(* CODESYS project CtaAppFU_1.0.0.2.library
   Description: FU Library der CTA
   Version: 1.0.0.2
   Title: CtaAppFU
   Author: SIS
   DocFormat: reStructuredText
   LanguageModelAttribute: qualified-access-only
   Placeholder: CtaAppFU
   DefaultNamespace: CtaAppFU
   CompiledLibraryCompatibilityVersion: CODESYS V3.5 SP16 Patch 3
   Company: CTA

Project tree, tasks and I/O mapping:
  libraries: Standard, 3.5.18.0 (System); CtaAppBasic, 1.0.0.0 (CTA); CtaAppBmk, 1.0.0.0 (CTA); CtaAppReport, 1.0.0.2 (CTA); CtaSysConfig, 1.0.0.2 (CTA); VisuDialogs, 3.5.16.20 (System); VisuSymbols, 4.5.0.0 (System); CtaSysFU, 1.0.0.0 (CTA); CtaAppTime, 1.0.0.1 (CTA); CtaVisSymbols, 1.0.0.0 (CTA); CtaAppInfluxLog, 1.0.0.0 (CTA); CtaSysBase, 1.0.0.0 (CTA); CtaAppWagoModbus, 1.0.0.0 (CTA); CtaAppModbus, 1.0.0.0 (CTA)
  40 Visualizations/
    ABB/
      580/
        visualisation DIA_ABB580
        TABLE/
          visualisation VIS_FU_ABB_TABLE
        VISU/
          visualisation VIS_ABB580
          visualisation VIS_ABB580_QUERY
      880/
        TABLE/
          visualisation VIS_FU_ABB_TABLE_880
        VISU/
          visualisation VIS_ABB880
          visualisation VIS_ABB880_QUERY
        visualisation DIA_ABB880
    BITZER/
      CSV/
        TABLE/
          visualisation VIS_FU_BITZER_TABLE
        VISU/
          visualisation VIS_BITZER_CSV
          visualisation VIS_BITZER_CSV_QUERY
        visualisation DIA_BITZER_CSV
  00000000-0000-0000-0000-000000000000|D:\CoDeSys\LibrariesV3\trunk\Intern\CAA\CAA Template\3.4.0.0 draft\Placeholder.xml
  00000000-0000-0000-0000-000000000000|D:\CoDeSys\LibrariesV3\trunk\Intern\CAA\CAA Template\3.2.0.3 draft\Prefix.pdf
  00000000-0000-0000-0000-000000000000|D:\CoDeSys\LibrariesV3\trunk\Intern\CAA\CAA Template\3.5.2.0 draft\Placeholder.xml
  20 Structs/
    Modbus/
      data type scParameter
      data type scModBus
    ABB/
      580/
        data type scFuAbb580Table
      880/
        data type scFuAbb880Table
    BITZER/
      CSV/
        data type enEnvelopeZone
        data type enEnvelopeState
        data type scFuBitzerCSVTable
        data type enFuState
  50 Images/
  10 Documenation/
    global variables VersionHistory
    global variables readMe
  21 Interface/
    ABB/
      880/
        interface ITF_FU_ABB_880: proayscTable
      580/
        interface ITF_FU_ABB_580: proayscTable
    BITZER/
      CSV/
        interface ITF_FU_BITZER_CSV: proayscTable
  11 Library Parameter/
    global variables Parameter
  12 Konstanten/
    global variables GlobalKonstant
  60 Textlisten/
    ABB 580/
      text list Error_ABB580_880
      text list Info_ABB580_880
      text list Warnung_ABB580_880
      text list FU_ABB_580_880_PARA
    BITZER/
      text list Error_BITZER_CSV
      text list Info_BITZER_CSV
      text list Warnung_BITZER_CSV
      text list FU_BITZER_CSV_PARA
  13 Globale Variablen/
    global variables GVL_FU
  text list GlobalTextList
  5ce3da45-db07-42e7-a21c-a00fff4ed8f6|C:\Users\sis\Downloads\dip-switch.svg
  5ce3da45-db07-42e7-a21c-a00fff4ed8f6|C:\Users\sis\Downloads\lightning-bolt-circle.svg
  30 Program Organization Units/
    ABB/
      580/
        function block FB_FU_ABB580 [ST]: proFU_TYPE, FB_INIT, COM_DATA, actCwSw, metParIdToMbAdr, metHzScaleFromFU, metHzScaleToFU, actCheckFirmWare, actCheckLastComCall, actTrendLog, actReport, actConfig, actTable, proayscTable
      880/
        function block FB_FU_ABB880 [ST]: FB_INIT, proFU_TYPE, COM_DATA, actCwSw, metParIdToMbAdr, metHzScaleFromFU, metHzScaleToFU, actCheckFirmWare, actCheckLastComCall, actTrendLog, actReport, actConfig, actTable, proayscTable
    Bitzer/
      CSV/
        function block FB_FU_BITZER_CSV [ST]: FB_INIT, COM_DATA, actCwSw, actCheckFirmWare, actCheckLastComCall, actTrendLog, actReport, actConfig, actTable, proayscTable, proFU_TYPE
  5ce3da45-db07-42e7-a21c-a00fff4ed8f6|C:\Users\sis\Downloads\sine-wave.svg
  5ce3da45-db07-42e7-a21c-a00fff4ed8f6|C:\Users\sis\Downloads\eye.svg
  5ce3da45-db07-42e7-a21c-a00fff4ed8f6|C:\Users\sis\Downloads\lan.svg
*)

// 20 Structs/Modbus/scParameter
TYPE scParameter :
	STRUCT
		scModBus	:	scModBus;
	END_STRUCT
END_TYPE

// 20 Structs/Modbus/scModBus
TYPE scModBus :
	STRUCT
		fbxMbErrorAsWarning	:	CtaSysConfig.fbBOOL;
	END_STRUCT
END_TYPE

// 20 Structs/ABB/580/scFuAbb580Table
TYPE scFuAbb580Table :
	STRUCT
		stParaNr		:	STRING(5);
		stValue			:	STRING(20);
	END_STRUCT
END_TYPE

// 20 Structs/ABB/880/scFuAbb880Table
TYPE scFuAbb880Table :
	STRUCT
		stParaNr		:	STRING(5);
		stValue			:	STRING(20);
	END_STRUCT
END_TYPE

// 20 Structs/BITZER/CSV/enEnvelopeZone
{attribute 'to_string'}
TYPE enEnvelopeZone :
	(
		inside 				:= 	0,
		SST_Low_SDT_Low		:=	1,
		SST_Low				:=	2,
		SST_Low_SDT_High	:=	3,
		SDT_High			:=	4,
		SST_High_SDT_High	:=	5,
		SST_High			:=	6,
		SST_High_SDT_Low	:=	7,
		SDT_Low				:= 	8	
	);
END_TYPE

// 20 Structs/BITZER/CSV/enEnvelopeState
{attribute 'to_string'}
TYPE enEnvelopeState :
	(
		stopped 	:= 0,
		starting 	:= 1,
		running		:= 2,
		stopping	:= 3,
		warning		:= 4,
		critical	:= 5,
		fault		:= 6,
		defrosting	:= 7
	);
END_TYPE

// 20 Structs/BITZER/CSV/scFuBitzerCSVTable
TYPE scFuBitzerCSVTable :
	STRUCT
		stParaNr		:	STRING(5);
		stValue			:	STRING(20);
	END_STRUCT
END_TYPE

// 20 Structs/BITZER/CSV/enFuState
{attribute 'to_string'}
TYPE enFuState :
	(
		not_ready		:=	0,
		power_not_ready :=	1,
		stopped			:=	2,
		short_Cycling	:=	3,
		start_Delay		:=	4,
		freeze			:=	5,
		running			:=	6,
		DC_Inj			:=	7,
		stopping		:=	8,
		locked			:=	9,
		fault			:= 10,
		service			:= 11
	);
END_TYPE

// 10 Documenation/VersionHistory
(* 

.. image:: ../../Images/CTA_Logo.jpg
   :align: right
   :width: 15% 

**Vorlage**   


============ =========== =========== ============================================
**Date**     **Version** **Author**  **Change**
------------ ----------- ----------- --------------------------------------------
04.03.2021   0.0.0.0     SIS         Vorlage erstellt

============ =========== =========== ============================================


*)
VAR_GLOBAL
    stInfo : STRING:= '0.0.0.0, Vorlage, CTA';
END_VAR

// 10 Documenation/readMe
(*

**ReadMe**
 
|	**Empfehlung**
|
|	Bibliothek CtaAppFU zur dämpfung und rampung von Signalen
|	Instanzieren Sie den CtaAppFU.fbFU in ihrem Funktionsbaustein oder POU beispielsweise als fbFUx ( x = Nr. des FU's 
|	Deklarieren Sie die Struktur Variable welche als Parameter und zur ansteuerung dienen wie im Code beispiel.
|  
| *Beispiel* 

+-----------------------+---------------------------------------------------------------------------------------------------------------------------------------------------------------------------------------------------------------------------------------------------------------------------------------------------------------------------------------------------------------------------------------------------------------------------------------+
| Beschreibung          |  Code                                                                                                                                                                                                                                                                                                                                                                                                                                 |
+=======================+=======================================================================================================================================================================================================================================================================================================================================================================================================================================+
| POU oder SmFb         | .. code-block:: codesys                                                                                                                                                                                                                                                                                                                                                                                                               |
|                       |                                                                                                                                                                                                                                                                                                                                                                                                                                       |
|                       |	// Deklaration als VAR im POU oder dem selbsterstellten Funktionsbaustein                                                                                                                                                                                                                                                                                                                                                        	|
|                       |   VAR   																																																				 																																																				|
|						|	    (*Frequenzumformer 1*)																																																		 																																																	|
|						|		fbFU1			: CtaAppFU.fbFU;																																																																																																|
|			 			|	END_VAR                                                                                                                                                                                                                                                                                                                                                                                                                          	|
+-----------------------+---------------------------------------------------------------------------------------------------------------------------------------------------------------------------------------------------------------------------------------------------------------------------------------------------------------------------------------------------------------------------------------------------------------------------------------+
| Code für Init         | .. code-block:: codesys                                                                                                                                                                                                                                                                                                                                                                                                               |
|                       |   																																																					 																																																				|
|			 			|	// Kopieren des nachfolgenden Codes in eine Action zur Initialisierung der Parameter. Zum Beispiel actConfig.																																																				 																										|
|                       |	{region "Parameter Temperaturfühler 1"}                                                                                                                                                                                                                                                                                                                                                                                             |
|			 			|		(*Basis*)                                                                                                                                                                                                                                                                                                                                                                                                                       |
|						|		fbFU1.scParameter.scModBus.fbxMbErrorAsWarning					(_WertInit := FALSE																	 	 		);     //P1 Parameter zur behandlung eines ModBus Fehlers als Warnung.																																															|
|						|	{endregion}                                                                                                                                                      																																																																    | 
|						|																																																																																																										|
+-----------------------+---------------------------------------------------------------------------------------------------------------------------------------------------------------------------------------------------------------------------------------------------------------------------------------------------------------------------------------------------------------------------------------------------------------------------------------+
*)                                                                                                                                                                                                                                                                                                                                                                                                                                                               
VAR_GLOBAL
	xReadMeDone              :   BOOL; 
END_VAR

// 13 Globale Variablen/GVL_FU
{attribute 'qualified_only'}
VAR_GLOBAL

END_VAR

// 11 Library Parameter/Parameter
{attribute 'qualified_only'}
VAR_GLOBAL CONSTANT
 	stABB580_FirmWare	:	STRING(20) := '2.20.0.12';
	stABB880_FirmWare	:	STRING(20) := '3.46.0.03';
	stBITZER_FirmWare	:	STRING(20) := '2.15.0.10';
END_VAR

// 12 Konstanten/GlobalKonstant
{attribute 'qualified_only'}
VAR_GLOBAL CONSTANT 	
	stReportTextListErrorAbb580_880   	: CtaAppReport.stReportTextList := 'CtaAppFU.Error_ABB580_880';
	stReportTextListWarningAbb580_880 	: CtaAppReport.stReportTextList := 'CtaAppFU.Warnung_ABB580_880';
	stReportTextListInfoAbb580_880  	: CtaAppReport.stReportTextList := 'CtaAppFU.Info_ABB580_880';
	stReportTextListErrorBitzerCsv   	: CtaAppReport.stReportTextList := 'CtaAppFU.Error_BITZER_CSV';
	stReportTextListWarningBitzerCsv 	: CtaAppReport.stReportTextList := 'CtaAppFU.Warnung_BITZER_CSV';
	stReportTextListInfoBitzerCsv    	: CtaAppReport.stReportTextList := 'CtaAppFU.Info_BITZER_CSV';		
END_VAR

// 30 Program Organization Units/ABB/580/FB_FU_ABB580
FUNCTION_BLOCK FB_FU_ABB580 EXTENDS CtaSysFU.FB_FU_BASE IMPLEMENTS ITF_FU_ABB_580
VAR_INPUT
END_VAR
VAR_OUTPUT
END_VAR
VAR
	(* Case *)
	iCaseCw					: 	INT;
	(* BUS Controll *)
	xResetAfterInit 		:   BOOL	:= TRUE;
	{attribute 'displaymode':='hex'}
	wControllWord   		:   WORD;
    wSollwert       		:   WORD;
	{attribute 'displaymode':='hex'}
    wStateWord      		:   WORD;
    wIstwert        		:   WORD;	
	xLocRemError			:	BOOL;
	(* HZ Scale Faktor *)
	rScaleFaktorHzMax   	:   REAL;    
    rScaleFaktorHzMin   	:   REAL;
	(* Energy Zähler *)
	uiGWhCount  			:   UINT;
    uiMWhCount  			:   UINT;
    uiKWhCount  			:   UINT;      
	(* Code from FU *)
	{attribute 'displaymode':='hex'}
	wErrorAkt       		:   WORD;
	{attribute 'displaymode':='hex'}
	wErrorOld1      		:   WORD;     
	{attribute 'displaymode':='hex'}   
	wErrorOld2      		:   WORD;    
	rHzOnError				:	REAL; 
	rTempOnError			:	REAL;
	(* Report*)     	
	iError					: 	INT;    
    difor					:	DINT;                                                                    
    ayErrorReporter			:	ARRAY[20..25] OF CtaAppReport.fbReporter;
	ayWarningReporter		:	ARRAY[20..25] OF CtaAppReport.fbReporter;	
	(* Trend Log *)
	fbTrendrAmpere			:	CtaAppInfluxLog.FB_LOG_NODE_REAL;
	fbTrendrVolt			:	CtaAppInfluxLog.FB_LOG_NODE_REAL;
	fbTrendrHz				:	CtaAppInfluxLog.FB_LOG_NODE_REAL;
	fbTrendrkW				:	CtaAppInfluxLog.FB_LOG_NODE_REAL;
	fbTrendrTemperatur		:	CtaAppInfluxLog.FB_LOG_NODE_REAL;
	fbTrendxError			:	CtaAppInfluxLog.FB_LOG_NODE_BOOL;
	fbTrendrGwh				:	CtaAppInfluxLog.FB_LOG_NODE_REAL;
	fbTrendrMwh				:	CtaAppInfluxLog.FB_LOG_NODE_REAL;
	fbTrendrkwh				:	CtaAppInfluxLog.FB_LOG_NODE_REAL;
	(* Modbus *)
	stVendorName			:	STRING(20);
	stMajorMinorRevision	:	STRING(20);
	xFirmWareOK				:	BOOL;
	fbLastComDataCall		:	CtaAppTime.fbTimeMeasurement;
	ltLastComCall			:	LTIME;
	xAccesOk				:	BOOL;
	xModbusOk				:	BOOL;
	aywTempRead				:	ARRAY[0..16] OF WORD;
	(* Tabelle *)
	ayscTable				:	ARRAY[0..16] OF scFuAbb580Table;
	(* Config *)
	fbConfigFile			:	CtaSysConfig.fbConfigFile;	
	scParameter				:	scParameter;
END_VAR

(* Config *)
actConfig();
(* Check Firmware *)
actCheckFirmWare();
(* Check Last Acces *)
actCheckLastComCall();
(* Controll & State Word *)
actCwSw();
(* Trend Log *)
actTrendLog();
(* Table *)
actTable();
(* Report *)
actReport();

PROPERTY proFU_TYPE : STRING(20)
GET
proFU_TYPE := 'ABB 580';
END_GET
END_PROPERTY

//FB_Init ist immer implizit verfügbar und wird primär für die Initialisierung verwendet.
//Der Rückgabewert wird nicht ausgewertet. Für gezielte Einflussnahme können Sie
//die Methoden explizit deklarieren und darin mit dem Standard-Initialisierungscode 
//zusätzlichen Code bereitstellen. Sie können den Rückgabewert auswerten.
METHOD FB_Init: BOOL
VAR_INPUT    
bInitRetains: BOOL; // TRUE: Die Retain-Variablen werden initialisiert (Reset warm / Reset kalt)    
bInCopyCode: BOOL;  // TRUE: Die Instanz wird danach in den Kopiercode kopiert (Online-Change)
END_VAR
SUPER^.stVisuDiaName := 'CtaAppFU.DIA_ABB580';
END_METHOD

METHOD COM_DATA
VAR_INPUT
	ITF_MB_CLIENT		:	CtaSysBase.ITF_BASE;
END_VAR
VAR
	ITF_MB_CLIENT_WAGO	: 	CtaAppWagoModbus.ITF_MbClient;
	ITF_MB_CLIENT_CS	:	CtaAppModbus.ITF_CLIENT;
END_VAR
IF __QUERYINTERFACE(ITF_MB_CLIENT,ITF_MB_CLIENT_WAGO) THEN
	(* COM DATA Call *)
	fbLastComDataCall.Start();
	(* Client Info *)
	ITF_MB_CLIENT_WAGO.metITF_BMK(THIS^);
	stVendorName 				:= ITF_MB_CLIENT_WAGO.sVendorName;
	stMajorMinorRevision 		:= ITF_MB_CLIENT_WAGO.sMajorMinorRevision;
	xModbusOk 					:= ITF_MB_CLIENT_WAGO.proModBusOK;
	(*-Modbus Fc----------------------------------------------------------------------------------------Umrechnung------------------------------------------------------------------------------------------Kommentar-------*)
	(* Fc3 *)	
	ITF_MB_CLIENT_WAGO.metFc3ReadHoldingRegister		(metParIdToMbAdr(00,04),ADR(aywTempRead[ 0])	,1,0);	wStateWord					:= aywTempRead[ 0];														// Parameter 00.04 Adr.    3	Status Word
	ITF_MB_CLIENT_WAGO.metFc3ReadHoldingRegister		(metParIdToMbAdr(00,05),ADR(aywTempRead[ 1])	,1,0);	wIstwert					:= aywTempRead[ 1];														// Parameter 00.05 Adr.    4	Status Wert
	ITF_MB_CLIENT_WAGO.metFc3ReadHoldingRegister		(metParIdToMbAdr(01,06),ADR(aywTempRead[ 2])	,1,0);	rAcknowledge_Hz				:= metHzScaleFromFU(aywTempRead[ 2],rScaleFaktorHzMax);					// Parameter 01.06 Adr.  105	Aktuelle Hz							
	ITF_MB_CLIENT_WAGO.metFc3ReadHoldingRegister		(metParIdToMbAdr(01,07),ADR(aywTempRead[ 3])	,1,0);  rAmpere						:= TO_REAL(aywTempRead[ 3])	/ 10;										// Parameter 01.07 Adr.  106	Aktuelle Ampere                                                               									
	ITF_MB_CLIENT_WAGO.metFc3ReadHoldingRegister		(metParIdToMbAdr(01,13),ADR(aywTempRead[ 4])	,1,0);	rVolt						:= aywTempRead[ 4];														// Parameter 01.13 Adr.  112	Aktuelle Spannung                                                                                               									
	ITF_MB_CLIENT_WAGO.metFc3ReadHoldingRegister		(metParIdToMbAdr(01,14),ADR(aywTempRead[ 5])	,1,0);	rkWatt						:= TO_REAL(aywTempRead[ 5])	/ 10;										// Parameter 01.14 Adr.  113	Aktuelle Leistung kW
	ITF_MB_CLIENT_WAGO.metFc3ReadHoldingRegister		(metParIdToMbAdr(01,18),ADR(aywTempRead[ 6])	,1,0);	uiGWhCount					:= aywTempRead[ 6];														// Parameter 01.18 Adr.  117	Leistung GWh
	ITF_MB_CLIENT_WAGO.metFc3ReadHoldingRegister		(metParIdToMbAdr(01,19),ADR(aywTempRead[ 7])	,1,0);	uiMWhCount					:= aywTempRead[ 7];														// Parameter 01.19 Adr.  118	Leistung MWh	
	ITF_MB_CLIENT_WAGO.metFc3ReadHoldingRegister		(metParIdToMbAdr(01,20),ADR(aywTempRead[ 8])	,1,0);	uiKWhCount					:= TO_UINT(aywTempRead[ 8])  / 10;										// Parameter 01.20 Adr.  119	Leistung KWh	
	ITF_MB_CLIENT_WAGO.metFc3ReadHoldingRegister		(metParIdToMbAdr(04,01),ADR(aywTempRead[ 9])	,1,0);	wErrorAkt					:= aywTempRead[ 9];														// Parameter 04.01 Adr.  400	Aktueller Fehler
	ITF_MB_CLIENT_WAGO.metFc3ReadHoldingRegister		(metParIdToMbAdr(04,02),ADR(aywTempRead[10])	,1,0);	wErrorOld1					:= aywTempRead[10];														// Parameter 04.02 Adr.  401	Letzter Fehler
	ITF_MB_CLIENT_WAGO.metFc3ReadHoldingRegister		(metParIdToMbAdr(04,03),ADR(aywTempRead[11])	,1,0);	wErrorOld2					:= aywTempRead[11];														// Parameter 04.03 Adr.  402	Vorletzter Fehler
	ITF_MB_CLIENT_WAGO.metFc3ReadHoldingRegister		(metParIdToMbAdr(05,10),ADR(aywTempRead[12])	,1,0);	rTemperatur					:= aywTempRead[12];														// Parameter 05.10 Adr.  509	Temperatur
(* Modbusprobleme Parameter Existieren nicht mehr 14.10.2024 SIS *)
//	ITF_MB_CLIENT_WAGO.metFc3ReadHoldingRegister		(metParIdToMbAdr(05,81),ADR(aywTempRead[13])	,1,0);	rHzOnError					:= metHzScaleFromFU(aywTempRead[13],rScaleFaktorHzMax);					// Parameter 05.81 Adr.  580	Frequenz bei Fehler
//	ITF_MB_CLIENT_WAGO.metFc3ReadHoldingRegister		(metParIdToMbAdr(05,87),ADR(aywTempRead[14])	,1,0);	rTempOnError				:= aywTempRead[14];														// Parameter 05.87 Adr.  586	Temperatur bei Fehler
	
	ITF_MB_CLIENT_WAGO.metFc3ReadHoldingRegister		(metParIdToMbAdr(30,13),ADR(aywTempRead[15])	,1,0);	rScaleFaktorHzMin			:= metHzScaleFromFU(aywTempRead[15],rScaleFaktorHzMax);					// Parameter 30.13 Adr. 3012	Min Hz Skalierfaktor
	ITF_MB_CLIENT_WAGO.metFc3ReadHoldingRegister		(metParIdToMbAdr(46,02),ADR(aywTempRead[16])	,1,0);	rScaleFaktorHzMax			:= TO_REAL(aywTempRead[16])  / 10;										// Parameter 46.02 Adr. 4600	Max Hz Skalierfaktor
	                                                                                                                        		                                                    					
	(*  Fc16 *)                                                                                             	        														        					
	ITF_MB_CLIENT_WAGO.metFc16WriteHoldingRegisters	(metParIdToMbAdr(00,01),ADR(wControllWord)		,1,0);  																									// Parameter 00.01 Adr.   0	Controll Word
	ITF_MB_CLIENT_WAGO.metFc16WriteHoldingRegisters	(metParIdToMbAdr(00,02),ADR(wSollwert)			,1,0);  																									// Parameter 00.02 Adr.   1	Soll Wert
ELSIF __QUERYINTERFACE(ITF_MB_CLIENT,ITF_MB_CLIENT_CS) THEN
	(* COM DATA Call *)
	fbLastComDataCall.Start();
	ITF_MB_CLIENT_CS.CREATE_JOB	( 3, metParIdToMbAdr(00,04),ADR(aywTempRead[ 0])	,1);	wStateWord					:= aywTempRead[ 0];														// Parameter 00.04 Adr.    3	Status Word
	ITF_MB_CLIENT_CS.CREATE_JOB ( 3, metParIdToMbAdr(00,05),ADR(aywTempRead[ 1])	,1);	wIstwert					:= aywTempRead[ 1];														// Parameter 00.05 Adr.    4	Status Wert
	ITF_MB_CLIENT_CS.CREATE_JOB ( 3, metParIdToMbAdr(01,06),ADR(aywTempRead[ 2])	,1);	rAcknowledge_Hz				:= metHzScaleFromFU(aywTempRead[ 2],rScaleFaktorHzMax);					// Parameter 01.06 Adr.  105	Aktuelle Hz							
	ITF_MB_CLIENT_CS.CREATE_JOB ( 3, metParIdToMbAdr(01,07),ADR(aywTempRead[ 3])	,1);  	rAmpere						:= TO_REAL(aywTempRead[ 3])	/ 10;										// Parameter 01.07 Adr.  106	Aktuelle Ampere                                  
	ITF_MB_CLIENT_CS.CREATE_JOB ( 3, metParIdToMbAdr(01,13),ADR(aywTempRead[ 4])	,1);	rVolt						:= aywTempRead[ 4];														// Parameter 01.13 Adr.  112	Aktuelle Spannung                                
	ITF_MB_CLIENT_CS.CREATE_JOB ( 3, metParIdToMbAdr(01,14),ADR(aywTempRead[ 5])	,1);	rkWatt						:= TO_REAL(aywTempRead[ 5])	/ 10;										// Parameter 01.14 Adr.  113	Aktuelle Leistung kW
	ITF_MB_CLIENT_CS.CREATE_JOB	( 3, metParIdToMbAdr(01,18),ADR(aywTempRead[ 6])	,1);	uiGWhCount					:= aywTempRead[ 6];														// Parameter 01.18 Adr.  117	Leistung GWh
	ITF_MB_CLIENT_CS.CREATE_JOB	( 3, metParIdToMbAdr(01,19),ADR(aywTempRead[ 7])	,1);	uiMWhCount					:= aywTempRead[ 7];														// Parameter 01.19 Adr.  118	Leistung MWh	
	ITF_MB_CLIENT_CS.CREATE_JOB	( 3, metParIdToMbAdr(01,20),ADR(aywTempRead[ 8])	,1);	uiKWhCount					:= TO_UINT(aywTempRead[ 8])  / 10;										// Parameter 01.20 Adr.  119	Leistung KWh	
	ITF_MB_CLIENT_CS.CREATE_JOB	( 3, metParIdToMbAdr(04,01),ADR(aywTempRead[ 9])	,1);	wErrorAkt					:= aywTempRead[ 9];														// Parameter 04.01 Adr.  400	Aktueller Fehler
	ITF_MB_CLIENT_CS.CREATE_JOB	( 3, metParIdToMbAdr(04,02),ADR(aywTempRead[10])	,1);	wErrorOld1					:= aywTempRead[10];														// Parameter 04.02 Adr.  401	Letzter Fehler
	ITF_MB_CLIENT_CS.CREATE_JOB	( 3, metParIdToMbAdr(04,03),ADR(aywTempRead[11])	,1);	wErrorOld2					:= aywTempRead[11];														// Parameter 04.03 Adr.  402	Vorletzter Fehler
	ITF_MB_CLIENT_CS.CREATE_JOB	( 3, metParIdToMbAdr(05,10),ADR(aywTempRead[12])	,1);	rTemperatur					:= aywTempRead[12];														// Parameter 05.10 Adr.  509	Temperatur
(* Modbusprobleme Parameter Existieren nicht mehr 14.10.2024 SIS *)
//	ITF_MB_CLIENT_CS.CREATE_JOB	( 3, metParIdToMbAdr(05,81),ADR(aywTempRead[13])	,1);	rHzOnError					:= metHzScaleFromFU(aywTempRead[13],rScaleFaktorHzMax);					// Parameter 05.81 Adr.  580	Frequenz bei Fehler
//	ITF_MB_CLIENT_CS.CREATE_JOB	( 3, metParIdToMbAdr(05,87),ADR(aywTempRead[14])	,1);	rTempOnError				:= aywTempRead[14];														// Parameter 05.87 Adr.  586	Temperatur bei Fehler
	
	ITF_MB_CLIENT_CS.CREATE_JOB	( 3, metParIdToMbAdr(30,13),ADR(aywTempRead[15])	,1);	rScaleFaktorHzMin			:= metHzScaleFromFU(aywTempRead[15],rScaleFaktorHzMax);					// Parameter 30.13 Adr. 3012	Min Hz Skalierfaktor
	ITF_MB_CLIENT_CS.CREATE_JOB	( 3, metParIdToMbAdr(46,02),ADR(aywTempRead[16])	,1);	rScaleFaktorHzMax			:= TO_REAL(aywTempRead[16])  / 10;										// Parameter 46.02 Adr. 4600	Max Hz Skalierfaktor

	(*  Fc16 *)                                                                                             	        														        					
	ITF_MB_CLIENT_CS.CREATE_JOB	(16, metParIdToMbAdr(00,01),ADR(wControllWord)		,1);  																									// Parameter 00.01 Adr.   0	Controll Word
	ITF_MB_CLIENT_CS.CREATE_JOB	(16, metParIdToMbAdr(00,02),ADR(wSollwert)			,1);  				
	xModbusOk := NOT ITF_MB_CLIENT_CS.ERROR;
	stVendorName := 'ABB';
	stMajorMinorRevision := Parameter.stABB580_FirmWare;
ELSE
	xModbusOk := FALSE;	
END_IF
xBusOK := xModbusOk;
END_METHOD

ACTION actCwSw:
(*--Controll Word-------------------------------------------State Word-----------------*)(*          
    wControllWord.0  = Aus1                                 wStateWord.0      = RDY_ON       
    wControllWord.1  = Aus2                                 wStateWord.1      = RDY_RUN      
    wControllWord.2  = Aus3                                 wStateWord.2      = RDY_REF      
    wControllWord.3  = Inhibit_Operation                    wStateWord.3      = TRIPPED      
    wControllWord.4  = Rampenausgang_Null                   wStateWord.4      = OFF_2_STATUS 
    wControllWord.5  = Rampenausgang_Halten                 wStateWord.5      = OFF_3_STATUS 
    wControllWord.6  = Rampeneingang_Null                   wStateWord.6      = SWC_ON_INHIB 
    wControllWord.7  = Quittierung                          wStateWord.7      = ALARM        
    wControllWord.8  = Jogging_1                            wStateWord.8      = AUF_SOLLWERT 
    wControllWord.9  = Jogginng_2                           wStateWord.9      = REMOTE       
    wControllWord.10 = Fernsteuerung                        wStateWord.10     = ÜBER_LIMIT   
    wControllWord.11 = EXT_CTRL_LOC                         wStateWord.11     = USER_0       
    wControllWord.12 = USER_0                               wStateWord.12     = USER_1       
    wControllWord.13 = USER_1                               wStateWord.13     = USER_2       
    wControllWord.14 = USER_2                               wStateWord.14     = USER_3       
    wControllWord.15 = USER_3                             	wStateWord.15     = RESERVE *)   
    
	   (* Quittieren *)
		wControllWord.7 := wStateWord.9 AND (xResetAfterInit 	 OR (ayErrorReporter[20].metGetQuitt() 
																 OR  ayErrorReporter[21].metGetQuitt() 
																 OR  ayErrorReporter[22].metGetQuitt() 
																 OR  ayErrorReporter[23].metGetQuitt()
																 OR  ayErrorReporter[24].metGetQuitt()
																 OR  ayErrorReporter[25].metGetQuitt()) 
																 OR xQuitt); 
		(* Status Werte *)
		xReady          := wStateWord.1 AND wStateWord.9;
		IF NOT xResetAfterInit THEN
			xLocRemError    := NOT wStateWord.9;
			xHandLockal		:= xLocRemError;
			xAcknowledge    := wStateWord.8; // OR wStateWord0616.14
			xError      	:= wStateWord.3;   
		END_IF;
		(* Bei Störmeldung oder Initialisierung in Case 0 Springen *)   
		IF xError THEN
			iCaseCw         := 0;   
		END_IF;   
		IF xReady THEN
			xResetAfterInit := FALSE;
		END_IF;
		(* Sollwert *)
		wSollwert := INT_TO_WORD(LIMIT(WORD_TO_INT(metHzScaleToFU(rScaleFaktorHzMin,rScaleFaktorHzMax)),WORD_TO_INT(metHzScaleToFU(rRelease_Hz,rScaleFaktorHzMax)),WORD_TO_INT(metHzScaleToFU(rScaleFaktorHzMax,rScaleFaktorHzMax)))); 
		(* FU Steuerung *)
		CASE iCaseCw OF
			0: // Nicht Einschaltbereit
				// Start Value 
				wControllWord.1  := TRUE;       // Nicht Aus 2 
				wControllWord.2  := TRUE;       // Nicht Aus 3 
				wControllWord.3  := FALSE;
				wControllWord.10 := TRUE;       // Steuerung Bus
				// Statusabfrage Nicht Einschaltbereit 
				wControllWord.0 := FALSE; 
				iCaseCw := iCaseCw + 1;   
			1: // Einschaltbereit           
				IF NOT wStateWord.1 AND NOT wStateWord.0 THEN      
					wControllWord.0 := FALSE;   
				ELSIF wStateWord.0 THEN 
					wControllWord.0 := TRUE; 
				END_IF;
				IF wStateWord.1 AND wStateWord.0 THEN                      
					iCaseCw := iCaseCw + 1;        
				END_IF;          
			2: // Betriebsbereit
				IF NOT xRelease AND NOT wStateWord.1 THEN
					iCaseCw := 0;
				END_IF;
				// Freigabe
				wControllWord.3 := xRelease;        
				// Wenn Betrieb Freigegeben weiter
				IF wStateWord.2 THEN
					IF wControllWord.3 THEN
						wControllWord.4 := TRUE;
						wControllWord.5 := TRUE;
						wControllWord.6 := TRUE;
						iCaseCw := iCaseCw + 1; 
					ELSE
						iCaseCw := 1;
					END_IF;
				END_IF;
			3: // Betrieb Freigegeben
				// Freigabe
				wControllWord.3 := xRelease AND iError = 0; 
				wControllWord.0 := xRelease AND iError = 0; 
				IF wControllWord.3 THEN
					wControllWord.4 := TRUE;
					wControllWord.5 := TRUE;
					wControllWord.6 := TRUE;
				ELSE
					iCaseCw := 0;
				END_IF;  
		ELSE
			iCaseCw := 0;           
		END_CASE;
END_ACTION

METHOD PRIVATE metParIdToMbAdr : WORD
VAR_INPUT
    usiMainParaId   :   USINT;
    usiSubParaId    :   USINT;
END_VAR
metParIdToMbAdr := (usiMainParaId * 100) + usiSubParaId - 1;
END_METHOD

METHOD PRIVATE metHzScaleFromFU : REAL
VAR_INPUT
    wModBusValue   :    WORD;
    rScaleFaktor   :    REAL;
END_VAR
VAR
	iModBusValue	:	INT;
END_VAR
iModBusValue := TO_INT(wModBusValue);
metHzScaleFromFU := rScaleFaktor / 20000 * TO_REAL(iModBusValue);
END_METHOD

METHOD PRIVATE metHzScaleToFU : WORD
VAR_INPUT
    rValue         :    REAL;
    rScaleFaktor   :    REAL;
END_VAR
rScaleFaktor := LIMIT(0,rScaleFaktor,65535);
IF rScaleFaktor <> 0 THEN
    metHzScaleToFU := TO_WORD(TO_INT(20000 / rScaleFaktor * rValue));
ELSE
    metHzScaleToFU := 0;
END_IF;
END_METHOD

ACTION actCheckFirmWare:
(* Check Firmware *)
IF FIND(stVendorName,'ABB') <> 0 THEN
	IF FIND(stMajorMinorRevision,Parameter.stABB580_FirmWare) <> 0 THEN
		xFirmWareOK := TRUE;	
	ELSE
		xFirmWareOK := FALSE;
	END_IF
ELSE
	xFirmWareOK := FALSE;
END_IF
END_ACTION

ACTION actCheckLastComCall:
(* Last Acces *)
ltLastComCall := fbLastComDataCall.Stop();
IF ltLastComCall <= LTIME#2S AND ltLastComCall >LTIME#0NS THEN
	xAccesOk := TRUE;
ELSE
	xAccesOk := FALSE;	
END_IF;
END_ACTION

ACTION actTrendLog:
(* Ampere *)
fbTrendrAmpere.ENABLE			:= TRUE;
fbTrendrAmpere.KEY				:= CONCAT(stObjID,'_rAmpere');
fbTrendrAmpere.SET_VALUE		:= rAmpere;

(* Volt *)
fbTrendrVolt.ENABLE				:= TRUE;
fbTrendrVolt.KEY				:= CONCAT(stObjID,'_rVolt');
fbTrendrVolt.SET_VALUE			:= rVolt;

(* HZ *)
fbTrendrHz.ENABLE				:= TRUE;
fbTrendrHz.KEY					:= CONCAT(stObjID,'_rHZ');
fbTrendrHz.SET_VALUE			:= rAcknowledge_Hz;

(* kW *)
fbTrendrkW.ENABLE				:= TRUE;
fbTrendrkW.KEY					:= CONCAT(stObjID,'_rkW');
fbTrendrkW.SET_VALUE			:= rkWatt;

(* Temperatur *)
fbTrendrTemperatur.ENABLE		:= TRUE;
fbTrendrTemperatur.KEY			:= CONCAT(stObjID,'_rTemperatur');
fbTrendrTemperatur.SET_VALUE	:= rTemperatur;

(* Error *)
fbTrendxError.ENABLE			:= TRUE;
fbTrendxError.KEY				:= CONCAT(stObjID,'_xError');
fbTrendxError.SET_VALUE			:= xError;

(* Gwh *)
fbTrendrGwh.ENABLE				:= TRUE;
fbTrendrGwh.KEY					:= CONCAT(stObjID,'_rGwh');
fbTrendrGwh.SET_VALUE			:= uiGWhCount;

(* Mwh *)
fbTrendrMwh.ENABLE				:= TRUE;
fbTrendrMwh.KEY					:= CONCAT(stObjID,'_rMwh');
fbTrendrMwh.SET_VALUE			:= uiMWhCount;

(* kwh *)
fbTrendrkwh.ENABLE				:= TRUE;
fbTrendrkwh.KEY					:= CONCAT(stObjID,'_rkwh');
fbTrendrkwh.SET_VALUE			:= uiKWhCount;
END_ACTION

ACTION actReport:
IF __QUERYINTERFACE(ITF_REPORTMANAGER,ITF_REPORTMANAGER) THEN

(* Errors *)                        
	(* Meldung Modbus Error *)
	ayErrorReporter[20].proPrio  := 1;
	ayErrorReporter[20].metReport(     		xSetReportIn					:= NOT xModbusOk AND xEnable,
											iReportID						:= 20,
											enReportTypeIn					:= SEL(scParameter.scModBus.fbxMbErrorAsWarning.xValue,CtaAppReport.enReportType.Error,CtaAppReport.enReportType.Warning),  
											enReportAcknowledgeTypeIn   	:= CtaAppReport.enReportacknowledgeType.Auto,
											tDelay							:= T#4S, 
											ITF_BMK_IN						:= THIS^,			              
											pstReportTextListIn				:= ADR(GlobalKonstant.stReportTextListErrorAbb580_880),
											stOptionalReportText		    := '',   
											iRetryTilReportLock 		    := 0, 
											xResetCount         		    := FALSE,  
											tReset						    := T#24H); 		

	(* Meldung Modbus Software Zugriff Fehler *)
	ayErrorReporter[21].proPrio  := 1;
	ayErrorReporter[21].metReport(     		xSetReportIn					:= NOT xAccesOk AND xEnable,
											iReportID						:= 21,
											enReportTypeIn					:= SEL(scParameter.scModBus.fbxMbErrorAsWarning.xValue,CtaAppReport.enReportType.Error,CtaAppReport.enReportType.Warning),  
											enReportAcknowledgeTypeIn   	:= CtaAppReport.enReportacknowledgeType.Auto,
											tDelay							:= T#4S, 
											ITF_BMK_IN						:= THIS^,			              
											pstReportTextListIn				:= ADR(GlobalKonstant.stReportTextListErrorAbb580_880),
											stOptionalReportText		    := '',   
											iRetryTilReportLock 		    := 0, 
											xResetCount         		    := FALSE,  
											tReset						    := T#24H); 		

	(* Meldung FU Error *)
	ayErrorReporter[22].proPrio  := 1;
	ayErrorReporter[22].metReport(     		xSetReportIn					:= xError AND xEnable,
											iReportID						:= 22,
											enReportTypeIn					:= CtaAppReport.enReportType.Error,  
											enReportAcknowledgeTypeIn   	:= CtaAppReport.enReportacknowledgeType.QUIT,
											tDelay							:= T#4S, 
											ITF_BMK_IN						:= THIS^,			              
											pstReportTextListIn				:= ADR(GlobalKonstant.stReportTextListErrorAbb580_880),
											stOptionalReportText		    := CtaAppReport.fcWordToHexString(wErrorAkt),   
											iRetryTilReportLock 		    := 0, 
											xResetCount         		    := FALSE,  
											tReset						    := T#24H); 	
											
	(* Meldung Firmware Missmatch *)
	ayWarningReporter[20].proPrio  := 1;
	ayWarningReporter[20].metReport(     	xSetReportIn					:= NOT xFirmWareOK AND xEnable,
											iReportID						:= 20,
											enReportTypeIn					:= CtaAppReport.enReportType.Warning,  
											enReportAcknowledgeTypeIn   	:= CtaAppReport.enReportacknowledgeType.Auto,
											tDelay							:= T#4S, 
											ITF_BMK_IN						:= THIS^,			              
											pstReportTextListIn				:= ADR(GlobalKonstant.stReportTextListWarningAbb580_880),
											stOptionalReportText		    := Parameter.stABB580_FirmWare,   
											iRetryTilReportLock 		    := 0, 
											xResetCount         		    := FALSE,  
											tReset						    := T#24H); 	
											
	(* Sync Reports *)                                         
	FOR difor := LOWER_BOUND(ayErrorReporter,1) TO UPPER_BOUND(ayErrorReporter,1) DO
		ITF_REPORTMANAGER.metSyncReporter(ayErrorReporter[difor]);	
	END_FOR;
	FOR difor := LOWER_BOUND(ayWarningReporter,1) TO UPPER_BOUND(ayWarningReporter,1) DO
		ITF_REPORTMANAGER.metSyncReporter(ayWarningReporter[difor]);	
	END_FOR;


END_IF;
END_ACTION

ACTION actConfig:
fbConfigFile();

scParameter.scModBus.fbxMbErrorAsWarning(_usiParaNr	:= 1, itfConfigFb := fbConfigFile);
END_ACTION

ACTION actTable:
ayscTable[00].stParaNr	:= 	'00.04';
ayscTable[00].stValue	:=	TO_STRING(CtaAppReport.fcWordToHexString(wStateWord));

ayscTable[01].stParaNr	:= 	'00.05';
ayscTable[01].stValue	:=	TO_STRING(wIstwert);

ayscTable[02].stParaNr	:= 	'01.06';
ayscTable[02].stValue	:=	CONCAT(TO_STRING(rAcknowledge_Hz),' Hz');

ayscTable[03].stParaNr	:= 	'01.07';
ayscTable[03].stValue	:=	CONCAT(TO_STRING(rAmpere),' A');

ayscTable[04].stParaNr	:= 	'01.13';
ayscTable[04].stValue	:=	CONCAT(TO_STRING(rVolt),' V');

ayscTable[05].stParaNr	:= 	'01.14';
ayscTable[05].stValue	:=	CONCAT(TO_STRING(rkWatt),' kW');

ayscTable[06].stParaNr	:= 	'01.18';
ayscTable[06].stValue	:=	CONCAT(TO_STRING(uiGWhCount),' GWh');

ayscTable[07].stParaNr	:= 	'01.19';
ayscTable[07].stValue	:=	CONCAT(TO_STRING(uiMWhCount),' MWh');

ayscTable[08].stParaNr	:= 	'01.20';
ayscTable[08].stValue	:=	CONCAT(TO_STRING(uiKWhCount),' KWh');

ayscTable[09].stParaNr	:= 	'04.01';
ayscTable[09].stValue	:=	TO_STRING(CtaAppReport.fcWordToHexString(wErrorAkt));

ayscTable[10].stParaNr	:= 	'04.02';
ayscTable[10].stValue	:=	TO_STRING(CtaAppReport.fcWordToHexString(wErrorOld1));

ayscTable[11].stParaNr	:= 	'04.03';
ayscTable[11].stValue	:=	TO_STRING(CtaAppReport.fcWordToHexString(wErrorOld2));

ayscTable[12].stParaNr	:= 	'05.10';
ayscTable[12].stValue	:=	CONCAT(TO_STRING(rTemperatur),' °C');

ayscTable[13].stParaNr	:= 	'05.81';
ayscTable[13].stValue	:=	CONCAT(TO_STRING(rHzOnError),' Hz');

ayscTable[14].stParaNr	:= 	'05.87';
ayscTable[14].stValue	:=	CONCAT(TO_STRING(rTempOnError),' °C');

ayscTable[15].stParaNr	:= 	'30.13';
ayscTable[15].stValue	:=	CONCAT(TO_STRING(rScaleFaktorHzMin),' Hz');

ayscTable[16].stParaNr	:= 	'46.02';
ayscTable[16].stValue	:=	CONCAT(TO_STRING(rScaleFaktorHzMax),' Hz');
END_ACTION

PROPERTY proayscTable : ARRAY[0..16] OF scFuAbb580Table;
GET
proayscTable := ayscTable;
END_GET
END_PROPERTY

END_FUNCTION_BLOCK

// 21 Interface/ABB/580/ITF_FU_ABB_580
INTERFACE ITF_FU_ABB_580 EXTENDS CtaSysFU.ITF_FU_BASE

PROPERTY proayscTable : ARRAY[0..16] OF scFuAbb580Table;
GET
END_GET
END_PROPERTY

END_INTERFACE

// 30 Program Organization Units/ABB/880/FB_FU_ABB880
FUNCTION_BLOCK FB_FU_ABB880 EXTENDS CtaSysFU.FB_FU_BASE IMPLEMENTS ITF_FU_ABB_880
VAR_INPUT
END_VAR
VAR_OUTPUT
END_VAR
VAR
	(* Case *)
	iCaseCw					: 	INT;
	(* BUS Controll *)
	xResetAfterInit 		:   BOOL	:= TRUE;
	{attribute 'displaymode':='hex'}
	wControllWord   		:   WORD;
    wSollwert       		:   WORD;
	{attribute 'displaymode':='hex'}
    wStateWord      		:   WORD;
    wIstwert        		:   WORD;	
	xLocRemError			:	BOOL;
	(* HZ Scale Faktor *)
	rScaleFaktorHzMax   	:   REAL;    
    rScaleFaktorHzMin   	:   REAL;
	(* Energy Zähler *)
	uiGWhCount  			:   UINT;
    uiMWhCount  			:   UINT;
    uiKWhCount  			:   UINT;      
	(* Code from FU *)
	{attribute 'displaymode':='hex'}
	wErrorAkt       		:   WORD;
	{attribute 'displaymode':='hex'}
	wErrorOld1      		:   WORD;     
	{attribute 'displaymode':='hex'}   
	wErrorOld2      		:   WORD;    
	rHzOnError				:	REAL; 
	rTempOnError			:	REAL;
	(* Report*)     	
	iError					: 	INT;    
    difor					:	DINT;                                                                    
    ayErrorReporter			:	ARRAY[20..25] OF CtaAppReport.fbReporter;
	ayWarningReporter		:	ARRAY[20..25] OF CtaAppReport.fbReporter;	
	(* Trend Log *)
    fbTrendrAmpere			:	CtaAppInfluxLog.FB_LOG_NODE_REAL;
	fbTrendrVolt			:	CtaAppInfluxLog.FB_LOG_NODE_REAL;
	fbTrendrHz				:	CtaAppInfluxLog.FB_LOG_NODE_REAL;
	fbTrendrkW				:	CtaAppInfluxLog.FB_LOG_NODE_REAL;
	fbTrendrTemperatur		:	CtaAppInfluxLog.FB_LOG_NODE_REAL;
	fbTrendxError			:	CtaAppInfluxLog.FB_LOG_NODE_BOOL;
	fbTrendrGwh				:	CtaAppInfluxLog.FB_LOG_NODE_REAL;
	fbTrendrMwh				:	CtaAppInfluxLog.FB_LOG_NODE_REAL;
	fbTrendrkwh				:	CtaAppInfluxLog.FB_LOG_NODE_REAL;
	(* Modbus *)
	stVendorName			:	STRING(20);
	stMajorMinorRevision	:	STRING(20);
	xFirmWareOK				:	BOOL;
	fbLastComDataCall		:	CtaAppTime.fbTimeMeasurement;
	ltLastComCall			:	LTIME;
	xAccesOk				:	BOOL;
	xModbusOk				:	BOOL;
	aywTempRead				:	ARRAY[0..16] OF WORD;
	(* Tabelle *)
	ayscTable				:	ARRAY[0..16] OF scFuAbb880Table;
	(* Config *)
	fbConfigFile			:	CtaSysConfig.fbConfigFile;	
	scParameter				:	scParameter;
END_VAR

(* Config *)
actConfig();
(* Check Firmware *)
actCheckFirmWare();
(* Check Last Acces *)
actCheckLastComCall();
(* Controll & State Word *)
actCwSw();
(* Trend Log *)
actTrendLog();
(* Table *)
actTable();
(* Report *)
actReport();

//FB_Init ist immer implizit verfügbar und wird primär für die Initialisierung verwendet.
//Der Rückgabewert wird nicht ausgewertet. Für gezielte Einflussnahme können Sie
//die Methoden explizit deklarieren und darin mit dem Standard-Initialisierungscode 
//zusätzlichen Code bereitstellen. Sie können den Rückgabewert auswerten.
METHOD FB_Init: BOOL
VAR_INPUT    
bInitRetains: BOOL; // TRUE: Die Retain-Variablen werden initialisiert (Reset warm / Reset kalt)    
bInCopyCode: BOOL;  // TRUE: Die Instanz wird danach in den Kopiercode kopiert (Online-Change)
END_VAR
SUPER^.stVisuDiaName := 'CtaAppFU.DIA_ABB880';
END_METHOD

PROPERTY proFU_TYPE : STRING(20)
GET
proFU_TYPE := 'ABB 880';
END_GET
END_PROPERTY

METHOD COM_DATA
VAR_INPUT
	ITF_MB_CLIENT		:	CtaSysBase.ITF_BASE;
END_VAR
VAR
	ITF_MB_CLIENT_WAGO	: 	CtaAppWagoModbus.ITF_MbClient;
	ITF_MB_CLIENT_CS	:	CtaAppModbus.ITF_CLIENT;
END_VAR
IF __QUERYINTERFACE(ITF_MB_CLIENT,ITF_MB_CLIENT_WAGO) THEN
	(* COM DATA Call *)
	fbLastComDataCall.Start();
	(* Client Info *)
	ITF_MB_CLIENT_WAGO.metITF_BMK(THIS^);
	stVendorName 				:= ITF_MB_CLIENT_WAGO.sVendorName;
	stMajorMinorRevision 		:= ITF_MB_CLIENT_WAGO.sMajorMinorRevision;
	xModbusOk 					:= ITF_MB_CLIENT_WAGO.proModBusOK;
	(*-Modbus Fc----------------------------------------------------------------------------------------Umrechnung------------------------------------------------------------------------------------------Kommentar-------*)
	(* Fc3 *)	
	ITF_MB_CLIENT_WAGO.metFc3ReadHoldingRegister		(metParIdToMbAdr(00,04),ADR(aywTempRead[ 0])	,1,0);	wStateWord					:= aywTempRead[ 0];														// Parameter 00.04 Adr.    3	Status Word
	ITF_MB_CLIENT_WAGO.metFc3ReadHoldingRegister		(metParIdToMbAdr(00,05),ADR(aywTempRead[ 1])	,1,0);	wIstwert					:= aywTempRead[ 1];														// Parameter 00.05 Adr.    4	Status Wert
	ITF_MB_CLIENT_WAGO.metFc3ReadHoldingRegister		(metParIdToMbAdr(01,06),ADR(aywTempRead[ 2])	,1,0);	rAcknowledge_Hz				:= metHzScaleFromFU(aywTempRead[ 2],rScaleFaktorHzMax);					// Parameter 01.06 Adr.  105	Aktuelle Hz							
	ITF_MB_CLIENT_WAGO.metFc3ReadHoldingRegister		(metParIdToMbAdr(01,07),ADR(aywTempRead[ 3])	,1,0);  rAmpere						:= TO_REAL(aywTempRead[ 3])	/ 10;										// Parameter 01.07 Adr.  106	Aktuelle Ampere                                                               									
	ITF_MB_CLIENT_WAGO.metFc3ReadHoldingRegister		(metParIdToMbAdr(01,13),ADR(aywTempRead[ 4])	,1,0);	rVolt						:= aywTempRead[ 4];														// Parameter 01.13 Adr.  112	Aktuelle Spannung                                                                                               									
	ITF_MB_CLIENT_WAGO.metFc3ReadHoldingRegister		(metParIdToMbAdr(01,14),ADR(aywTempRead[ 5])	,1,0);	rkWatt						:= TO_REAL(aywTempRead[ 5])	/ 10;										// Parameter 01.14 Adr.  113	Aktuelle Leistung kW
	ITF_MB_CLIENT_WAGO.metFc3ReadHoldingRegister		(metParIdToMbAdr(01,18),ADR(aywTempRead[ 6])	,1,0);	uiGWhCount					:= aywTempRead[ 6];														// Parameter 01.18 Adr.  117	Leistung GWh
	ITF_MB_CLIENT_WAGO.metFc3ReadHoldingRegister		(metParIdToMbAdr(01,19),ADR(aywTempRead[ 7])	,1,0);	uiMWhCount					:= aywTempRead[ 7];														// Parameter 01.19 Adr.  118	Leistung MWh	
	ITF_MB_CLIENT_WAGO.metFc3ReadHoldingRegister		(metParIdToMbAdr(01,20),ADR(aywTempRead[ 8])	,1,0);	uiKWhCount					:= TO_UINT(aywTempRead[ 8])  / 10;										// Parameter 01.20 Adr.  119	Leistung KWh	
	ITF_MB_CLIENT_WAGO.metFc3ReadHoldingRegister		(metParIdToMbAdr(04,01),ADR(aywTempRead[ 9])	,1,0);	wErrorAkt					:= aywTempRead[ 9];														// Parameter 04.01 Adr.  400	Aktueller Fehler
	ITF_MB_CLIENT_WAGO.metFc3ReadHoldingRegister		(metParIdToMbAdr(04,02),ADR(aywTempRead[10])	,1,0);	wErrorOld1					:= aywTempRead[10];														// Parameter 04.02 Adr.  401	Letzter Fehler
	ITF_MB_CLIENT_WAGO.metFc3ReadHoldingRegister		(metParIdToMbAdr(04,03),ADR(aywTempRead[11])	,1,0);	wErrorOld2					:= aywTempRead[11];														// Parameter 04.03 Adr.  402	Vorletzter Fehler
	ITF_MB_CLIENT_WAGO.metFc3ReadHoldingRegister		(metParIdToMbAdr(05,10),ADR(aywTempRead[12])	,1,0);	rTemperatur					:= aywTempRead[12];														// Parameter 05.10 Adr.  509	Temperatur
(* Modbusprobleme Parameter Existieren nicht mehr 14.10.2024 SIS *)
//	ITF_MB_CLIENT_WAGO.metFc3ReadHoldingRegister		(metParIdToMbAdr(05,81),ADR(aywTempRead[13])	,1,0);	rHzOnError					:= metHzScaleFromFU(aywTempRead[13],rScaleFaktorHzMax);					// Parameter 05.81 Adr.  580	Frequenz bei Fehler
//	ITF_MB_CLIENT_WAGO.metFc3ReadHoldingRegister		(metParIdToMbAdr(05,87),ADR(aywTempRead[14])	,1,0);	rTempOnError				:= aywTempRead[14];														// Parameter 05.87 Adr.  586	Temperatur bei Fehler
	
	ITF_MB_CLIENT_WAGO.metFc3ReadHoldingRegister		(metParIdToMbAdr(30,13),ADR(aywTempRead[15])	,1,0);	rScaleFaktorHzMin			:= metHzScaleFromFU(aywTempRead[15],rScaleFaktorHzMax);					// Parameter 30.13 Adr. 3012	Min Hz Skalierfaktor
	ITF_MB_CLIENT_WAGO.metFc3ReadHoldingRegister		(metParIdToMbAdr(46,02),ADR(aywTempRead[16])	,1,0);	rScaleFaktorHzMax			:= TO_REAL(aywTempRead[16])  / 10;										// Parameter 46.02 Adr. 4600	Max Hz Skalierfaktor
	                                                                                                                        		                                                    					
	(*  Fc16 *)                                                                                             	        														        					
	ITF_MB_CLIENT_WAGO.metFc16WriteHoldingRegisters	(metParIdToMbAdr(00,01),ADR(wControllWord)		,1,0);  																									// Parameter 00.01 Adr.   0	Controll Word
	ITF_MB_CLIENT_WAGO.metFc16WriteHoldingRegisters	(metParIdToMbAdr(00,02),ADR(wSollwert)			,1,0);  																									// Parameter 00.02 Adr.   1	Soll Wert
ELSIF __QUERYINTERFACE(ITF_MB_CLIENT,ITF_MB_CLIENT_CS) THEN
	(* COM DATA Call *)
	fbLastComDataCall.Start();
	ITF_MB_CLIENT_CS.CREATE_JOB	( 3, metParIdToMbAdr(00,04),ADR(aywTempRead[ 0])	,1);	wStateWord					:= aywTempRead[ 0];														// Parameter 00.04 Adr.    3	Status Word
	ITF_MB_CLIENT_CS.CREATE_JOB ( 3, metParIdToMbAdr(00,05),ADR(aywTempRead[ 1])	,1);	wIstwert					:= aywTempRead[ 1];														// Parameter 00.05 Adr.    4	Status Wert
	ITF_MB_CLIENT_CS.CREATE_JOB ( 3, metParIdToMbAdr(01,06),ADR(aywTempRead[ 2])	,1);	rAcknowledge_Hz				:= metHzScaleFromFU(aywTempRead[ 2],rScaleFaktorHzMax);					// Parameter 01.06 Adr.  105	Aktuelle Hz							
	ITF_MB_CLIENT_CS.CREATE_JOB ( 3, metParIdToMbAdr(01,07),ADR(aywTempRead[ 3])	,1);  	rAmpere						:= TO_REAL(aywTempRead[ 3])	/ 10;										// Parameter 01.07 Adr.  106	Aktuelle Ampere                                  
	ITF_MB_CLIENT_CS.CREATE_JOB ( 3, metParIdToMbAdr(01,13),ADR(aywTempRead[ 4])	,1);	rVolt						:= aywTempRead[ 4];														// Parameter 01.13 Adr.  112	Aktuelle Spannung                                
	ITF_MB_CLIENT_CS.CREATE_JOB ( 3, metParIdToMbAdr(01,14),ADR(aywTempRead[ 5])	,1);	rkWatt						:= TO_REAL(aywTempRead[ 5])	/ 10;										// Parameter 01.14 Adr.  113	Aktuelle Leistung kW
	ITF_MB_CLIENT_CS.CREATE_JOB	( 3, metParIdToMbAdr(01,18),ADR(aywTempRead[ 6])	,1);	uiGWhCount					:= aywTempRead[ 6];														// Parameter 01.18 Adr.  117	Leistung GWh
	ITF_MB_CLIENT_CS.CREATE_JOB	( 3, metParIdToMbAdr(01,19),ADR(aywTempRead[ 7])	,1);	uiMWhCount					:= aywTempRead[ 7];														// Parameter 01.19 Adr.  118	Leistung MWh	
	ITF_MB_CLIENT_CS.CREATE_JOB	( 3, metParIdToMbAdr(01,20),ADR(aywTempRead[ 8])	,1);	uiKWhCount					:= TO_UINT(aywTempRead[ 8])  / 10;										// Parameter 01.20 Adr.  119	Leistung KWh	
	ITF_MB_CLIENT_CS.CREATE_JOB	( 3, metParIdToMbAdr(04,01),ADR(aywTempRead[ 9])	,1);	wErrorAkt					:= aywTempRead[ 9];														// Parameter 04.01 Adr.  400	Aktueller Fehler
	ITF_MB_CLIENT_CS.CREATE_JOB	( 3, metParIdToMbAdr(04,02),ADR(aywTempRead[10])	,1);	wErrorOld1					:= aywTempRead[10];														// Parameter 04.02 Adr.  401	Letzter Fehler
	ITF_MB_CLIENT_CS.CREATE_JOB	( 3, metParIdToMbAdr(04,03),ADR(aywTempRead[11])	,1);	wErrorOld2					:= aywTempRead[11];														// Parameter 04.03 Adr.  402	Vorletzter Fehler
	ITF_MB_CLIENT_CS.CREATE_JOB	( 3, metParIdToMbAdr(05,10),ADR(aywTempRead[12])	,1);	rTemperatur					:= aywTempRead[12];														// Parameter 05.10 Adr.  509	Temperatur
(* Modbusprobleme Parameter Existieren nicht mehr 14.10.2024 SIS *)
//	ITF_MB_CLIENT_CS.CREATE_JOB	( 3, metParIdToMbAdr(05,81),ADR(aywTempRead[13])	,1);	rHzOnError					:= metHzScaleFromFU(aywTempRead[13],rScaleFaktorHzMax);					// Parameter 05.81 Adr.  580	Frequenz bei Fehler
//	ITF_MB_CLIENT_CS.CREATE_JOB	( 3, metParIdToMbAdr(05,87),ADR(aywTempRead[14])	,1);	rTempOnError				:= aywTempRead[14];														// Parameter 05.87 Adr.  586	Temperatur bei Fehler
	
	ITF_MB_CLIENT_CS.CREATE_JOB	( 3, metParIdToMbAdr(30,13),ADR(aywTempRead[15])	,1);	rScaleFaktorHzMin			:= metHzScaleFromFU(aywTempRead[15],rScaleFaktorHzMax);					// Parameter 30.13 Adr. 3012	Min Hz Skalierfaktor
	ITF_MB_CLIENT_CS.CREATE_JOB	( 3, metParIdToMbAdr(46,02),ADR(aywTempRead[16])	,1);	rScaleFaktorHzMax			:= TO_REAL(aywTempRead[16])  / 10;										// Parameter 46.02 Adr. 4600	Max Hz Skalierfaktor

	(*  Fc16 *)                                                                                             	        														        					
	ITF_MB_CLIENT_CS.CREATE_JOB	(16, metParIdToMbAdr(00,01),ADR(wControllWord)		,1);  																									// Parameter 00.01 Adr.   0	Controll Word
	ITF_MB_CLIENT_CS.CREATE_JOB	(16, metParIdToMbAdr(00,02),ADR(wSollwert)			,1);  				
	xModbusOk := NOT ITF_MB_CLIENT_CS.ERROR;
	stVendorName := 'ABB';
	stMajorMinorRevision := Parameter.stABB580_FirmWare;
ELSE
	xModbusOk := FALSE;	
END_IF
xBusOK := xModbusOk;
END_METHOD

ACTION actCwSw:
(*--Controll Word-------------------------------------------State Word-----------------*)(*          
    wControllWord.0  = Aus1                                 wStateWord.0      = RDY_ON       
    wControllWord.1  = Aus2                                 wStateWord.1      = RDY_RUN      
    wControllWord.2  = Aus3                                 wStateWord.2      = RDY_REF      
    wControllWord.3  = Inhibit_Operation                    wStateWord.3      = TRIPPED      
    wControllWord.4  = Rampenausgang_Null                   wStateWord.4      = OFF_2_STATUS 
    wControllWord.5  = Rampenausgang_Halten                 wStateWord.5      = OFF_3_STATUS 
    wControllWord.6  = Rampeneingang_Null                   wStateWord.6      = SWC_ON_INHIB 
    wControllWord.7  = Quittierung                          wStateWord.7      = ALARM        
    wControllWord.8  = Jogging_1                            wStateWord.8      = AUF_SOLLWERT 
    wControllWord.9  = Jogginng_2                           wStateWord.9      = REMOTE       
    wControllWord.10 = Fernsteuerung                        wStateWord.10     = ÜBER_LIMIT   
    wControllWord.11 = EXT_CTRL_LOC                         wStateWord.11     = USER_0       
    wControllWord.12 = USER_0                               wStateWord.12     = USER_1       
    wControllWord.13 = USER_1                               wStateWord.13     = USER_2       
    wControllWord.14 = USER_2                               wStateWord.14     = USER_3       
    wControllWord.15 = USER_3                             	wStateWord.15     = RESERVE *)   
    
	   (* Quittieren *)
		wControllWord.7 := wStateWord.9 AND (xResetAfterInit 	 OR (ayErrorReporter[20].metGetQuitt() 
																 OR  ayErrorReporter[21].metGetQuitt() 
																 OR  ayErrorReporter[22].metGetQuitt() 
																 OR  ayErrorReporter[23].metGetQuitt()
																 OR  ayErrorReporter[24].metGetQuitt()
																 OR  ayErrorReporter[25].metGetQuitt()) 
																 OR xQuitt); 
		(* Status Werte *)
		xReady          := wStateWord.1 AND wStateWord.9;
		IF NOT xResetAfterInit THEN
			xLocRemError    := NOT wStateWord.9;
			xHandLockal		:= xLocRemError;
			xAcknowledge    := wStateWord.8; // OR wStateWord0616.14
			xError      	:= wStateWord.3;   
		END_IF;
		(* Bei Störmeldung oder Initialisierung in Case 0 Springen *)   
		IF xError THEN
			iCaseCw         := 0;   
		END_IF;   
		IF xReady THEN
			xResetAfterInit := FALSE;
		END_IF;
		(* Sollwert *)
		wSollwert := INT_TO_WORD(LIMIT(WORD_TO_INT(metHzScaleToFU(rScaleFaktorHzMin,rScaleFaktorHzMax)),WORD_TO_INT(metHzScaleToFU(rRelease_Hz,rScaleFaktorHzMax)),WORD_TO_INT(metHzScaleToFU(rScaleFaktorHzMax,rScaleFaktorHzMax)))); 
		(* FU Steuerung *)
		CASE iCaseCw OF
			0: // Nicht Einschaltbereit
				// Start Value 
				wControllWord.1  := TRUE;       // Nicht Aus 2 
				wControllWord.2  := TRUE;       // Nicht Aus 3 
				wControllWord.3  := FALSE;
				wControllWord.10 := TRUE;       // Steuerung Bus
				// Statusabfrage Nicht Einschaltbereit 
				wControllWord.0 := FALSE; 
				iCaseCw := iCaseCw + 1;   
			1: // Einschaltbereit           
				IF NOT wStateWord.1 AND NOT wStateWord.0 THEN      
					wControllWord.0 := FALSE;   
				ELSIF wStateWord.0 THEN 
					wControllWord.0 := TRUE; 
				END_IF;
				IF wStateWord.1 AND wStateWord.0 THEN                      
					iCaseCw := iCaseCw + 1;        
				END_IF;          
			2: // Betriebsbereit
				IF NOT xRelease AND NOT wStateWord.1 THEN
					iCaseCw := 0;
				END_IF;
				// Freigabe
				wControllWord.3 := xRelease;        
				// Wenn Betrieb Freigegeben weiter
				IF wStateWord.2 THEN
					IF wControllWord.3 THEN
						wControllWord.4 := TRUE;
						wControllWord.5 := TRUE;
						wControllWord.6 := TRUE;
						iCaseCw := iCaseCw + 1; 
					ELSE
						iCaseCw := 1;
					END_IF;
				END_IF;
			3: // Betrieb Freigegeben
				// Freigabe
				wControllWord.3 := xRelease AND iError = 0; 
				wControllWord.0 := xRelease AND iError = 0; 
				IF wControllWord.3 THEN
					wControllWord.4 := TRUE;
					wControllWord.5 := TRUE;
					wControllWord.6 := TRUE;
				ELSE
					iCaseCw := 0;
				END_IF;  
		ELSE
			iCaseCw := 0;           
		END_CASE;
END_ACTION

METHOD PRIVATE metParIdToMbAdr : WORD
VAR_INPUT
    usiMainParaId   :   USINT;
    usiSubParaId    :   USINT;
END_VAR
metParIdToMbAdr := (usiMainParaId * 100) + usiSubParaId - 1;
END_METHOD

METHOD PRIVATE metHzScaleFromFU : REAL
VAR_INPUT
    wModBusValue   :    WORD;
    rScaleFaktor   :    REAL;
END_VAR
VAR
	iModBusValue	:	INT;
END_VAR
iModBusValue := TO_INT(wModBusValue);
metHzScaleFromFU := rScaleFaktor / 20000 * TO_REAL(iModBusValue);
END_METHOD

METHOD PRIVATE metHzScaleToFU : WORD
VAR_INPUT
    rValue         :    REAL;
    rScaleFaktor   :    REAL;
END_VAR
rScaleFaktor := LIMIT(0,rScaleFaktor,65535);
IF rScaleFaktor <> 0 THEN
    metHzScaleToFU := TO_WORD(TO_INT(20000 / rScaleFaktor * rValue));
ELSE
    metHzScaleToFU := 0;
END_IF;
END_METHOD

ACTION actCheckFirmWare:
(* Check Firmware *)
IF FIND(stVendorName,'ABB') <> 0 THEN
	IF FIND(stMajorMinorRevision,Parameter.stABB880_FirmWare) <> 0 THEN
		xFirmWareOK := TRUE;	
	ELSE
		xFirmWareOK := FALSE;
	END_IF
ELSE
	xFirmWareOK := FALSE;
END_IF
END_ACTION

ACTION actCheckLastComCall:
(* Last Acces *)
ltLastComCall := fbLastComDataCall.Stop();
IF ltLastComCall <= LTIME#2S AND ltLastComCall >LTIME#0NS THEN
	xAccesOk := TRUE;
ELSE
	xAccesOk := FALSE;	
END_IF;
END_ACTION

ACTION actTrendLog:
(* Ampere *)
fbTrendrAmpere.ENABLE			:= TRUE;
fbTrendrAmpere.KEY				:= CONCAT(stObjID,'_rAmpere');
fbTrendrAmpere.SET_VALUE		:= rAmpere;

(* Volt *)
fbTrendrVolt.ENABLE				:= TRUE;
fbTrendrVolt.KEY				:= CONCAT(stObjID,'_rVolt');
fbTrendrVolt.SET_VALUE			:= rVolt;

(* HZ *)
fbTrendrHz.ENABLE				:= TRUE;
fbTrendrHz.KEY					:= CONCAT(stObjID,'_rHZ');
fbTrendrHz.SET_VALUE			:= rAcknowledge_Hz;

(* kW *)
fbTrendrkW.ENABLE				:= TRUE;
fbTrendrkW.KEY					:= CONCAT(stObjID,'_rkW');
fbTrendrkW.SET_VALUE			:= rkWatt;

(* Temperatur *)
fbTrendrTemperatur.ENABLE		:= TRUE;
fbTrendrTemperatur.KEY			:= CONCAT(stObjID,'_rTemperatur');
fbTrendrTemperatur.SET_VALUE	:= rTemperatur;

(* Error *)
fbTrendxError.ENABLE			:= TRUE;
fbTrendxError.KEY				:= CONCAT(stObjID,'_xError');
fbTrendxError.SET_VALUE			:= xError;

(* Gwh *)
fbTrendrGwh.ENABLE				:= TRUE;
fbTrendrGwh.KEY					:= CONCAT(stObjID,'_rGwh');
fbTrendrGwh.SET_VALUE			:= uiGWhCount;

(* Mwh *)
fbTrendrMwh.ENABLE				:= TRUE;
fbTrendrMwh.KEY					:= CONCAT(stObjID,'_rMwh');
fbTrendrMwh.SET_VALUE			:= uiMWhCount;

(* kwh *)
fbTrendrkwh.ENABLE				:= TRUE;
fbTrendrkwh.KEY					:= CONCAT(stObjID,'_rkwh');
fbTrendrkwh.SET_VALUE			:= uiKWhCount;
END_ACTION

ACTION actReport:
IF __QUERYINTERFACE(ITF_REPORTMANAGER,ITF_REPORTMANAGER) THEN

(* Errors *)                        
	(* Meldung Modbus Error *)
	ayErrorReporter[20].proPrio  := 1;
	ayErrorReporter[20].metReport(     		xSetReportIn					:= NOT xModbusOk AND xEnable,
											iReportID						:= 20,
											enReportTypeIn					:= SEL(scParameter.scModBus.fbxMbErrorAsWarning.xValue,CtaAppReport.enReportType.Error,CtaAppReport.enReportType.Warning),  
											enReportAcknowledgeTypeIn   	:= CtaAppReport.enReportacknowledgeType.Auto,
											tDelay							:= T#4S, 
											ITF_BMK_IN						:= THIS^,			              
											pstReportTextListIn				:= ADR(GlobalKonstant.stReportTextListErrorAbb580_880),
											stOptionalReportText		    := '',   
											iRetryTilReportLock 		    := 0, 
											xResetCount         		    := FALSE,  
											tReset						    := T#24H); 		

	(* Meldung Modbus Software Zugriff Fehler *)
	ayErrorReporter[21].proPrio  := 1;
	ayErrorReporter[21].metReport(     		xSetReportIn					:= NOT xAccesOk AND xEnable,
											iReportID						:= 21,
											enReportTypeIn					:= SEL(scParameter.scModBus.fbxMbErrorAsWarning.xValue,CtaAppReport.enReportType.Error,CtaAppReport.enReportType.Warning),  
											enReportAcknowledgeTypeIn   	:= CtaAppReport.enReportacknowledgeType.Auto,
											tDelay							:= T#4S, 
											ITF_BMK_IN						:= THIS^,			              
											pstReportTextListIn				:= ADR(GlobalKonstant.stReportTextListErrorAbb580_880),
											stOptionalReportText		    := '',   
											iRetryTilReportLock 		    := 0, 
											xResetCount         		    := FALSE,  
											tReset						    := T#24H); 		

	(* Meldung FU Error *)
	ayErrorReporter[22].proPrio  := 1;
	ayErrorReporter[22].metReport(     		xSetReportIn					:= xError AND xEnable,
											iReportID						:= 22,
											enReportTypeIn					:= CtaAppReport.enReportType.Error,  
											enReportAcknowledgeTypeIn   	:= CtaAppReport.enReportacknowledgeType.QUIT,
											tDelay							:= T#4S, 
											ITF_BMK_IN						:= THIS^,			              
											pstReportTextListIn				:= ADR(GlobalKonstant.stReportTextListErrorAbb580_880),
											stOptionalReportText		    := CtaAppReport.fcWordToHexString(wErrorAkt),   
											iRetryTilReportLock 		    := 0, 
											xResetCount         		    := FALSE,  
											tReset						    := T#24H); 	
											
	(* Meldung Firmware Missmatch *)
	ayWarningReporter[20].proPrio  := 1;
	ayWarningReporter[20].metReport(     	xSetReportIn					:= NOT xFirmWareOK AND xEnable,
											iReportID						:= 20,
											enReportTypeIn					:= CtaAppReport.enReportType.Warning,  
											enReportAcknowledgeTypeIn   	:= CtaAppReport.enReportacknowledgeType.Auto,
											tDelay							:= T#4S, 
											ITF_BMK_IN						:= THIS^,			              
											pstReportTextListIn				:= ADR(GlobalKonstant.stReportTextListWarningAbb580_880),
											stOptionalReportText		    := Parameter.stABB580_FirmWare,   
											iRetryTilReportLock 		    := 0, 
											xResetCount         		    := FALSE,  
											tReset						    := T#24H); 	
											
	(* Sync Reports *)                                         
	FOR difor := LOWER_BOUND(ayErrorReporter,1) TO UPPER_BOUND(ayErrorReporter,1) DO
		ITF_REPORTMANAGER.metSyncReporter(ayErrorReporter[difor]);	
	END_FOR;
	FOR difor := LOWER_BOUND(ayWarningReporter,1) TO UPPER_BOUND(ayWarningReporter,1) DO
		ITF_REPORTMANAGER.metSyncReporter(ayWarningReporter[difor]);	
	END_FOR;


END_IF;
END_ACTION

ACTION actConfig:
fbConfigFile();

scParameter.scModBus.fbxMbErrorAsWarning(_usiParaNr	:= 1, itfConfigFb := fbConfigFile);
END_ACTION

ACTION actTable:
ayscTable[00].stParaNr	:= 	'00.04';
ayscTable[00].stValue	:=	TO_STRING(CtaAppReport.fcWordToHexString(wStateWord));

ayscTable[01].stParaNr	:= 	'00.05';
ayscTable[01].stValue	:=	TO_STRING(wIstwert);

ayscTable[02].stParaNr	:= 	'01.06';
ayscTable[02].stValue	:=	CONCAT(TO_STRING(rAcknowledge_Hz),' Hz');

ayscTable[03].stParaNr	:= 	'01.07';
ayscTable[03].stValue	:=	CONCAT(TO_STRING(rAmpere),' A');

ayscTable[04].stParaNr	:= 	'01.13';
ayscTable[04].stValue	:=	CONCAT(TO_STRING(rVolt),' V');

ayscTable[05].stParaNr	:= 	'01.14';
ayscTable[05].stValue	:=	CONCAT(TO_STRING(rkWatt),' kW');

ayscTable[06].stParaNr	:= 	'01.18';
ayscTable[06].stValue	:=	CONCAT(TO_STRING(rkWatt),' GWh');

ayscTable[07].stParaNr	:= 	'01.19';
ayscTable[07].stValue	:=	CONCAT(TO_STRING(rkWatt),' MWh');

ayscTable[08].stParaNr	:= 	'01.20';
ayscTable[08].stValue	:=	CONCAT(TO_STRING(rkWatt),' KWh');

ayscTable[09].stParaNr	:= 	'04.01';
ayscTable[09].stValue	:=	TO_STRING(CtaAppReport.fcWordToHexString(wErrorAkt));

ayscTable[10].stParaNr	:= 	'04.02';
ayscTable[10].stValue	:=	TO_STRING(CtaAppReport.fcWordToHexString(wErrorOld1));

ayscTable[11].stParaNr	:= 	'04.03';
ayscTable[11].stValue	:=	TO_STRING(CtaAppReport.fcWordToHexString(wErrorOld2));

ayscTable[12].stParaNr	:= 	'05.10';
ayscTable[12].stValue	:=	CONCAT(TO_STRING(rTemperatur),' °C');

ayscTable[13].stParaNr	:= 	'05.81';
ayscTable[13].stValue	:=	CONCAT(TO_STRING(rHzOnError),' Hz');

ayscTable[14].stParaNr	:= 	'05.87';
ayscTable[14].stValue	:=	CONCAT(TO_STRING(rTempOnError),' °C');

ayscTable[15].stParaNr	:= 	'30.13';
ayscTable[15].stValue	:=	CONCAT(TO_STRING(rScaleFaktorHzMin),' Hz');

ayscTable[16].stParaNr	:= 	'46.02';
ayscTable[16].stValue	:=	CONCAT(TO_STRING(rScaleFaktorHzMax),' Hz');
END_ACTION

PROPERTY proayscTable : ARRAY[0..16] OF scFuAbb880Table;
GET
proayscTable := ayscTable;
END_GET
END_PROPERTY

END_FUNCTION_BLOCK

// 21 Interface/ABB/880/ITF_FU_ABB_880
INTERFACE ITF_FU_ABB_880 EXTENDS CtaSysFU.ITF_FU_BASE

PROPERTY proayscTable : ARRAY[0..16] OF scFuAbb880Table;
GET
END_GET
END_PROPERTY

END_INTERFACE

// 30 Program Organization Units/Bitzer/CSV/FB_FU_BITZER_CSV
FUNCTION_BLOCK FB_FU_BITZER_CSV EXTENDS CtaSysFU.FB_FU_BASE IMPLEMENTS ITF_FU_BITZER_CSV
VAR_INPUT
END_VAR
VAR_OUTPUT
END_VAR
VAR
	(* BUS Controll *)
	xResetAfterInit 			:   BOOL	:= TRUE;
	{attribute 'displaymode':='hex'}
	wControllWord   			:   WORD;
    wSollwert       			:   WORD;
	{attribute 'displaymode':='hex'}
    wStateWord      			:   WORD;
    wIstwert        			:   WORD;
	(* Parameter *)
	siSollwertZuFu				:	SINT;
	uiMotordrehZahl				:	UINT;
	siOilTemperature			:	SINT;
	uiSuctionPreassure			:	UINT;
	uiDischargePreassure		:	UINT;
	siEvaporatingTemperature	:	SINT;
	siCondensingTemperature		:	SINT;
	uiEnvelopeStatus			:	enEnvelopeState;
	uiEnvelopeZone				:	enEnvelopeZone;
	siMotorTemperature			:	SINT;
	uiStatusState				:	enFuState;
	siIGBT_Temperatur			:	SINT;
	siColdPlateTemperature		:	SINT;
	
	(* HZ Scale Faktor *)
	rScaleFaktorHzMax   		:   REAL;    
    rScaleFaktorHzMin   		:   REAL;
	(* Energy Zähler *)
	uiGWhCount  				:   UINT;
    uiMWhCount  				:   UINT;
    uiKWhCount  				:   UINT;      
	(* Code from FU *)
	{attribute 'displaymode':='hex'}
	dwFaultWord       			:   DWORD;
	{attribute 'displaymode':='hex'}
	dwCriticalWord     			:   DWORD;     
	{attribute 'displaymode':='hex'}   
	dwWarningWord      			:   DWORD; 
	(* Report*)     	
	iError						: 	INT;    
    difor						:	DINT;                                                                    
    ayErrorReporter				:	ARRAY[20..25] OF CtaAppReport.fbReporter;
	ayWarningReporter			:	ARRAY[20..25] OF CtaAppReport.fbReporter;	
	(* Trend Log *)
	fbTrendrSollwert			:	CtaAppInfluxLog.FB_LOG_NODE_REAL;
	fbTrendrIstwert				:	CtaAppInfluxLog.FB_LOG_NODE_REAL;
	fbTrendrRPM					:	CtaAppInfluxLog.FB_LOG_NODE_REAL;
	fbTrendiOilTemp				:	CtaAppInfluxLog.FB_LOG_NODE_INT;
	fbTrendiSucPreassure		:	CtaAppInfluxLog.FB_LOG_NODE_INT;
	fbTrendiDisPreassure		:	CtaAppInfluxLog.FB_LOG_NODE_INT;
	fbTrendiEvapTemp			:	CtaAppInfluxLog.FB_LOG_NODE_INT;
	fbTrendiCondTemp			:	CtaAppInfluxLog.FB_LOG_NODE_INT;
	fbTrendiEnvStatus			:	CtaAppInfluxLog.FB_LOG_NODE_INT;
	fbTrendiEnvZone				:	CtaAppInfluxLog.FB_LOG_NODE_INT;
	fbTrendiMotorTemp			:	CtaAppInfluxLog.FB_LOG_NODE_INT;
	fbTrendiFuState				:	CtaAppInfluxLog.FB_LOG_NODE_INT;
	fbTrendiIgbtTemp			:	CtaAppInfluxLog.FB_LOG_NODE_INT;
	fbTrendiColdPlateTemp		:	CtaAppInfluxLog.FB_LOG_NODE_INT;
	fbTrendxError				:	CtaAppInfluxLog.FB_LOG_NODE_BOOL;
	(* Modbus *)
	stVendorName			:	STRING(20);
	stMajorMinorRevision	:	STRING(20);
	xFirmWareOK				:	BOOL;
	fbLastComDataCall		:	CtaAppTime.fbTimeMeasurement;
	ltLastComCall			:	LTIME;
	xAccesOk				:	BOOL;
	xModbusOk				:	BOOL;
	aywTempRead				:	ARRAY[0..17] OF WORD;
	(* Tabelle *)
	ayscTable				:	ARRAY[0..17] OF scFuBitzerCSVTable;
	(* Config *)
	fbConfigFile			:	CtaSysConfig.fbConfigFile;	
	scParameter				:	scParameter;
END_VAR

(* Config *)
actConfig();
(* Check Firmware *)
actCheckFirmWare();
(* Check Last Acces *)
actCheckLastComCall();
(* Controll & State Word *)
actCwSw();
(* Trend Log *)
actTrendLog();
(* Table *)
actTable();
(* Report *)
actReport();

//FB_Init ist immer implizit verfügbar und wird primär für die Initialisierung verwendet.
//Der Rückgabewert wird nicht ausgewertet. Für gezielte Einflussnahme können Sie
//die Methoden explizit deklarieren und darin mit dem Standard-Initialisierungscode 
//zusätzlichen Code bereitstellen. Sie können den Rückgabewert auswerten.
METHOD FB_Init: BOOL
VAR_INPUT    
bInitRetains: BOOL; // TRUE: Die Retain-Variablen werden initialisiert (Reset warm / Reset kalt)    
bInCopyCode: BOOL;  // TRUE: Die Instanz wird danach in den Kopiercode kopiert (Online-Change)
END_VAR
SUPER^.stVisuDiaName := 'CtaAppFU.DIA_BITZER_CSV';
END_METHOD

METHOD COM_DATA
VAR_INPUT
	ITF_MB_CLIENT		:	CtaSysBase.ITF_BASE;
END_VAR
VAR
	ITF_MB_CLIENT_WAGO	:	CtaAppWagoModbus.ITF_MbClient;
END_VAR
IF __QUERYINTERFACE(ITF_MB_CLIENT,ITF_MB_CLIENT_WAGO) THEN
	(* COM DATA Call *)
	fbLastComDataCall.Start();
	(* Client Info *)
	ITF_MB_CLIENT_WAGO.metITF_BMK(THIS^);
	stVendorName 				:= 'BITZER';							// BITZER unterstüzt FC43 nicht
	stMajorMinorRevision 		:= Parameter.stBITZER_FirmWare;
	xModbusOk 					:= ITF_MB_CLIENT_WAGO.proModBusOK;
	(*-Modbus Fc----------------------------------------------------------------------------------------Umrechnung------------------------------------------------------------------------------------------Kommentar-------*)
	(* Fc3 *)	
	ITF_MB_CLIENT_WAGO.metFc4ReadInputRegister		(100	,ADR(aywTempRead[ 0])	,1,0);	siSollwertZuFu				:= TO_SINT(aywTempRead[ 0]/100);											
	ITF_MB_CLIENT_WAGO.metFc3ReadHoldingRegister		(101	,ADR(aywTempRead[ 1])	,1,0);	wIstwert					:= aywTempRead[ 1];														
	ITF_MB_CLIENT_WAGO.metFc3ReadHoldingRegister		(103	,ADR(aywTempRead[ 2])	,1,0);	wStateWord					:= aywTempRead[ 2];														
	ITF_MB_CLIENT_WAGO.metFc3ReadHoldingRegister		(10001	,ADR(aywTempRead[ 3])	,1,0);	uiMotordrehZahl				:= TO_UINT(aywTempRead[ 3]);												
	ITF_MB_CLIENT_WAGO.metFc3ReadHoldingRegister		(11000	,ADR(aywTempRead[ 4])	,2,0);  dwFaultWord					:= aywTempRead[ 4];										                                                        									
	ITF_MB_CLIENT_WAGO.metFc3ReadHoldingRegister		(11002	,ADR(aywTempRead[ 5])	,2,0);	dwCriticalWord				:= aywTempRead[ 5];														                                                                                          									
	ITF_MB_CLIENT_WAGO.metFc3ReadHoldingRegister		(11004	,ADR(aywTempRead[ 6])	,2,0);	dwWarningWord				:= aywTempRead[ 6];										
	ITF_MB_CLIENT_WAGO.metFc3ReadHoldingRegister		(12000	,ADR(aywTempRead[ 7])	,1,0);	siOilTemperature			:= TO_SINT(aywTempRead[ 7]/10);														
	ITF_MB_CLIENT_WAGO.metFc3ReadHoldingRegister		(12001	,ADR(aywTempRead[ 8])	,1,0);	uiSuctionPreassure			:= aywTempRead[ 8]/100;														
	ITF_MB_CLIENT_WAGO.metFc3ReadHoldingRegister		(12002	,ADR(aywTempRead[ 9])	,1,0);	uiDischargePreassure		:= aywTempRead[ 9]/10;										
	ITF_MB_CLIENT_WAGO.metFc3ReadHoldingRegister		(12003	,ADR(aywTempRead[10])	,1,0);	siEvaporatingTemperature	:= TO_SINT(aywTempRead[10])/10;														
	ITF_MB_CLIENT_WAGO.metFc3ReadHoldingRegister		(12004	,ADR(aywTempRead[11])	,1,0);	siCondensingTemperature		:= TO_SINT(aywTempRead[11])/10;														
	ITF_MB_CLIENT_WAGO.metFc3ReadHoldingRegister		(12005	,ADR(aywTempRead[12])	,1,0);	uiEnvelopeStatus			:= aywTempRead[12];														
	ITF_MB_CLIENT_WAGO.metFc3ReadHoldingRegister		(12006	,ADR(aywTempRead[13])	,1,0);	uiEnvelopeZone				:= aywTempRead[13];														
	ITF_MB_CLIENT_WAGO.metFc3ReadHoldingRegister		(13000	,ADR(aywTempRead[14])	,1,0);	siMotorTemperature			:= TO_SINT(aywTempRead[14])/10;					
	ITF_MB_CLIENT_WAGO.metFc3ReadHoldingRegister		(14002	,ADR(aywTempRead[15])	,1,0);	uiStatusState				:= aywTempRead[15];														
	ITF_MB_CLIENT_WAGO.metFc3ReadHoldingRegister		(14100	,ADR(aywTempRead[16])	,1,0);	siIGBT_Temperatur			:= TO_SINT(aywTempRead[16])/10;					
	ITF_MB_CLIENT_WAGO.metFc3ReadHoldingRegister		(14101	,ADR(aywTempRead[17])	,1,0);	siColdPlateTemperature		:= TO_SINT(aywTempRead[17])/10;										

	(*  Fc16 *)                                                                                             	        														        					
	ITF_MB_CLIENT_WAGO.metFc6WriteHoldingRegister	(110,ADR(wControllWord)		,1,0);  																					
ELSE
	xModbusOk := FALSE;	
END_IF
xBusOK := xModbusOk;
END_METHOD

ACTION actCwSw:
(*--Controll Word-------------------------------------------State Word-----------------*)(*          
    wControllWord.0  = Reserviert                           wStateWord.0      = Nicht verwendet       
    wControllWord.1  = Reserviert                           wStateWord.1      = Frequenzumrichter bereit      
    wControllWord.2  = Reserviert                           wStateWord.2      = Betrieb freigegeben      
    wControllWord.3  = Betrieb freigeben                    wStateWord.3      = Störung     
    wControllWord.4  = Reserviert                 			wStateWord.4      = Nicht verwendet	 
    wControllWord.5  = Reserviert			                wStateWord.5      = Nicht verwendet 
    wControllWord.6  = Anlauf			                   	wStateWord.6      = Nicht verwendet 
    wControllWord.7  = Reset	                          	wStateWord.7      = Warnung        
    wControllWord.8  = Reserviert                           wStateWord.8      = Auf Sollwert 
    wControllWord.9  = Reserviert                           wStateWord.9      = Nicht verwendet       
    wControllWord.10 = Daten gültig                        	wStateWord.10     = Begrenzer aktiv   
    wControllWord.11 = Reserviert                         	wStateWord.11     = In Betrieb       
    wControllWord.12 = Reserviert                           wStateWord.12     = Anlauf aktiv       
    wControllWord.13 = Reserviert                           wStateWord.13     = Kritisch       
    wControllWord.14 = Reserviert                           wStateWord.14     = Nicht verwendet       
    wControllWord.15 = Reserviert                           wStateWord.15     = Nicht verwendet *)   
    
(* Quittieren *)
wControllWord.7 :=  (xResetAfterInit	OR (ayErrorReporter[20].metGetQuitt() 
										OR	ayErrorReporter[21].metGetQuitt() 
										OR	ayErrorReporter[22].metGetQuitt() 
										OR	ayErrorReporter[23].metGetQuitt()
										OR	ayErrorReporter[24].metGetQuitt()
										OR	ayErrorReporter[25].metGetQuitt()) 
										OR	xQuitt); 
(* Status Werte *)
xReady	:= wStateWord.1;

IF NOT xResetAfterInit THEN
	xAcknowledge    := wStateWord.11; 
	xError      	:= wStateWord.3;   
END_IF;

IF xReady THEN
	xResetAfterInit := FALSE;
END_IF;
END_ACTION

ACTION actCheckFirmWare:
(* Check Firmware *)
IF FIND(stVendorName,'BITZER') <> 0 THEN
	IF FIND(stMajorMinorRevision,Parameter.stBITZER_FirmWare) <> 0 THEN
		xFirmWareOK := TRUE;	
	ELSE
		xFirmWareOK := FALSE;
	END_IF
ELSE
	xFirmWareOK := FALSE;
END_IF
END_ACTION

ACTION actCheckLastComCall:
(* Last Acces *)
ltLastComCall := fbLastComDataCall.Stop();
IF ltLastComCall <= LTIME#2S AND ltLastComCall >LTIME#0NS THEN
	xAccesOk := TRUE;
ELSE
	xAccesOk := FALSE;	
END_IF;
END_ACTION

ACTION actTrendLog:
(* Sollwert *)
fbTrendrSollwert.ENABLE				:= TRUE;
fbTrendrSollwert.KEY				:= CONCAT(stObjID,' _%_Ist');
fbTrendrSollwert.SET_VALUE			:= siSollwertZuFu;

(* Istwert *)
fbTrendrIstwert.ENABLE				:= TRUE;
fbTrendrIstwert.KEY					:= CONCAT(stObjID,'_%_Soll');
fbTrendrIstwert.SET_VALUE			:= TO_REAL(wIstwert);

(* RPM *)
fbTrendrRPM.ENABLE					:= TRUE;
fbTrendrRPM.KEY						:= CONCAT(stObjID,'_RPM');
fbTrendrRPM.SET_VALUE				:= uiMotordrehZahl;

(* Öltemperatur *)
fbTrendiOilTemp.ENABLE				:= TRUE;
fbTrendiOilTemp.KEY					:= CONCAT(stObjID,'_°C_Oil');
fbTrendiOilTemp.SET_VALUE			:= siOilTemperature;

(* Verdampfungsdruck *)
fbTrendiSucPreassure.ENABLE			:= TRUE;
fbTrendiSucPreassure.KEY			:= CONCAT(stObjID,'_bar_To');
fbTrendiSucPreassure.SET_VALUE		:= TO_INT(uiSuctionPreassure);

(* Verflüssigungsdruck  *)
fbTrendiDisPreassure.ENABLE			:= TRUE;
fbTrendiDisPreassure.KEY			:= CONCAT(stObjID,'_bar_Tc');
fbTrendiDisPreassure.SET_VALUE		:= TO_INT(uiDischargePreassure);

(* Verdampfungstemperatur  *)
fbTrendiEvapTemp.ENABLE				:= TRUE;
fbTrendiEvapTemp.KEY				:= CONCAT(stObjID,'_°C_To');
fbTrendiEvapTemp.SET_VALUE			:= siEvaporatingTemperature;

(* Verflüssigungstemperatur  *)
fbTrendiCondTemp.ENABLE				:= TRUE;
fbTrendiCondTemp.KEY				:= CONCAT(stObjID,'_°C_Tc');
fbTrendiCondTemp.SET_VALUE			:= siCondensingTemperature;

(* Aktueller Status  *)
fbTrendiEnvStatus.ENABLE			:= TRUE;
fbTrendiEnvStatus.KEY				:= CONCAT(stObjID,' _EnvelopeState');
fbTrendiEnvStatus.SET_VALUE			:= uiEnvelopeStatus;

(* Status Einsatzgrenze *)
fbTrendiEnvZone.ENABLE				:= TRUE;
fbTrendiEnvZone.KEY					:= CONCAT(stObjID,'_EnvelopeZone');
fbTrendiEnvZone.SET_VALUE			:= uiEnvelopeZone;

(* Motortemperatur  *)
fbTrendiMotorTemp.ENABLE			:= TRUE;
fbTrendiMotorTemp.KEY				:= CONCAT(stObjID,'_°C_Motor');
fbTrendiMotorTemp.SET_VALUE			:= siMotorTemperature;

(* Status Frequenzumrichter  *)
fbTrendiFuState.ENABLE				:= TRUE;
fbTrendiFuState.KEY					:= CONCAT(stObjID,'_Status_FU');
fbTrendiFuState.SET_VALUE			:= uiStatusState;

(* IGBT Temperatur *)
fbTrendiIgbtTemp.ENABLE				:= TRUE;
fbTrendiIgbtTemp.KEY				:= CONCAT(stObjID,'_°C_IGBT');
fbTrendiIgbtTemp.SET_VALUE			:= siIGBT_Temperatur;

(* Kühlplatten Temperatur *)
fbTrendiColdPlateTemp.ENABLE		:= TRUE;
fbTrendiColdPlateTemp.KEY			:= CONCAT(stObjID,'_°C_Plate');
fbTrendiColdPlateTemp.SET_VALUE		:= siColdPlateTemperature;

(* Kühlplatten Temperatur *)
fbTrendxError.ENABLE				:= TRUE;
fbTrendxError.KEY					:= CONCAT(stObjID,'_xError');
fbTrendxError.SET_VALUE				:= xError;
END_ACTION

ACTION actReport:
IF __QUERYINTERFACE(ITF_REPORTMANAGER,ITF_REPORTMANAGER) THEN

(* Errors *)                        
	(* Meldung Modbus Error *)
	ayErrorReporter[20].proPrio  := 1;
	ayErrorReporter[20].metReport(     		xSetReportIn					:= NOT xModbusOk AND xEnable,
											iReportID						:= 20,
											enReportTypeIn					:= SEL(scParameter.scModBus.fbxMbErrorAsWarning.xValue,CtaAppReport.enReportType.Error,CtaAppReport.enReportType.Warning),  
											enReportAcknowledgeTypeIn   	:= CtaAppReport.enReportacknowledgeType.Auto,
											tDelay							:= T#4S, 
											ITF_BMK_IN						:= THIS^,			              
											pstReportTextListIn				:= ADR(GlobalKonstant.stReportTextListErrorBitzerCsv),
											stOptionalReportText		    := '',   
											iRetryTilReportLock 		    := 0, 
											xResetCount         		    := FALSE,  
											tReset						    := T#24H); 		

	(* Meldung Modbus Software Zugriff Fehler *)
	ayErrorReporter[21].proPrio  := 1;
	ayErrorReporter[21].metReport(     		xSetReportIn					:= NOT xAccesOk AND xEnable,
											iReportID						:= 21,
											enReportTypeIn					:= SEL(scParameter.scModBus.fbxMbErrorAsWarning.xValue,CtaAppReport.enReportType.Error,CtaAppReport.enReportType.Warning),  
											enReportAcknowledgeTypeIn   	:= CtaAppReport.enReportacknowledgeType.Auto,
											tDelay							:= T#4S, 
											ITF_BMK_IN						:= THIS^,			              
											pstReportTextListIn				:= ADR(GlobalKonstant.stReportTextListErrorBitzerCsv),
											stOptionalReportText		    := '',   
											iRetryTilReportLock 		    := 0, 
											xResetCount         		    := FALSE,  
											tReset						    := T#24H); 		

	(* Meldung FU Error *)
	ayErrorReporter[22].proPrio  := 1;
	ayErrorReporter[22].metReport(     		xSetReportIn					:= xError AND xEnable,
											iReportID						:= 22,
											enReportTypeIn					:= CtaAppReport.enReportType.Error,  
											enReportAcknowledgeTypeIn   	:= CtaAppReport.enReportacknowledgeType.QUIT,
											tDelay							:= T#4S, 
											ITF_BMK_IN						:= THIS^,			              
											pstReportTextListIn				:= ADR(GlobalKonstant.stReportTextListErrorBitzerCsv),
											stOptionalReportText		    := CtaAppReport.fcWordToHexString(TO_WORD(dwFaultWord)),   
											iRetryTilReportLock 		    := 0, 
											xResetCount         		    := FALSE,  
											tReset						    := T#24H); 	
											
	(* Meldung Firmware Missmatch *)
	ayWarningReporter[20].proPrio  := 1;
	ayWarningReporter[20].metReport(     	xSetReportIn					:= NOT xFirmWareOK AND xEnable,
											iReportID						:= 20,
											enReportTypeIn					:= CtaAppReport.enReportType.Warning,  
											enReportAcknowledgeTypeIn   	:= CtaAppReport.enReportacknowledgeType.Auto,
											tDelay							:= T#4S, 
											ITF_BMK_IN						:= THIS^,			              
											pstReportTextListIn				:= ADR(GlobalKonstant.stReportTextListWarningBitzerCsv),
											stOptionalReportText		    := Parameter.stABB580_FirmWare,   
											iRetryTilReportLock 		    := 0, 
											xResetCount         		    := FALSE,  
											tReset						    := T#24H); 	
											
	(* Sync Reports *)                                         
	FOR difor := LOWER_BOUND(ayErrorReporter,1) TO UPPER_BOUND(ayErrorReporter,1) DO
		ITF_REPORTMANAGER.metSyncReporter(ayErrorReporter[difor]);	
	END_FOR;
	FOR difor := LOWER_BOUND(ayWarningReporter,1) TO UPPER_BOUND(ayWarningReporter,1) DO
		ITF_REPORTMANAGER.metSyncReporter(ayWarningReporter[difor]);	
	END_FOR;


END_IF;
END_ACTION

ACTION actConfig:
fbConfigFile();

scParameter.scModBus.fbxMbErrorAsWarning(_usiParaNr	:= 1, itfConfigFb := fbConfigFile);
END_ACTION

ACTION actTable:
ayscTable[00].stParaNr	:=	'1';
ayscTable[00].stValue	:=	CONCAT(TO_STRING(siSollwertZuFu),' %');

ayscTable[01].stParaNr	:= 	'2';
ayscTable[01].stValue	:=	CONCAT(TO_STRING(wIstwert),' %');

ayscTable[02].stParaNr	:= 	'3';
ayscTable[02].stValue	:=	CONCAT(TO_STRING(uiMotordrehZahl),' RPM');

ayscTable[03].stParaNr	:= 	'4';
ayscTable[03].stValue	:=	TO_STRING(CtaAppReport.fcWordToHexString(wStateWord));

ayscTable[04].stParaNr	:= 	'5';
ayscTable[04].stValue	:=	TO_STRING(CtaAppReport.fcWordToHexString(TO_WORD(dwFaultWord)));

ayscTable[05].stParaNr	:= 	'6';
ayscTable[05].stValue	:=	TO_STRING(CtaAppReport.fcWordToHexString(TO_WORD(dwCriticalWord)));

ayscTable[06].stParaNr	:= 	'7';
ayscTable[06].stValue	:=	TO_STRING(CtaAppReport.fcWordToHexString(TO_WORD(dwWarningWord)));

ayscTable[07].stParaNr	:=	'8';
ayscTable[07].stValue	:=	TO_STRING(uiStatusState);

ayscTable[08].stParaNr	:= 	'9';
ayscTable[08].stValue	:=	TO_STRING(uiEnvelopeStatus);

ayscTable[09].stParaNr	:= 	'10';
ayscTable[09].stValue	:=	TO_STRING(uiEnvelopeZone);

ayscTable[10].stParaNr	:= 	'11';
ayscTable[10].stValue	:=	CONCAT(TO_STRING(uiSuctionPreassure),' bar');

ayscTable[11].stParaNr	:= 	'12';
ayscTable[11].stValue	:=	CONCAT(TO_STRING(siEvaporatingTemperature),' °C');

ayscTable[12].stParaNr	:= 	'13';
ayscTable[12].stValue	:=	CONCAT(TO_STRING(uiDischargePreassure),' bar');

ayscTable[13].stParaNr	:= 	'14';
ayscTable[13].stValue	:=	CONCAT(TO_STRING(siCondensingTemperature),' °C');

ayscTable[14].stParaNr	:= 	'15';
ayscTable[14].stValue	:=	CONCAT(TO_STRING(siOilTemperature),' °C');

ayscTable[15].stParaNr	:= 	'16';
ayscTable[15].stValue	:=	CONCAT(TO_STRING(siMotorTemperature),' °C');

ayscTable[16].stParaNr	:= '17';
ayscTable[16].stValue	:=	CONCAT(TO_STRING(siIGBT_Temperatur),' °C');

ayscTable[17].stParaNr	:=	'18';
ayscTable[17].stValue	:=	CONCAT(TO_STRING(siColdPlateTemperature),' °C');
END_ACTION

PROPERTY proayscTable : ARRAY[0..17] OF scFuBitzerCSVTable;
GET
proayscTable := ayscTable;
END_GET
END_PROPERTY

PROPERTY proFU_TYPE : STRING(20)
GET
proFU_TYPE := 'BITZER CSV';
END_GET
END_PROPERTY

END_FUNCTION_BLOCK

// 21 Interface/BITZER/CSV/ITF_FU_BITZER_CSV
INTERFACE ITF_FU_BITZER_CSV EXTENDS CtaSysFU.ITF_FU_BASE

PROPERTY proayscTable : ARRAY[0..17] OF scFuBitzerCSVTable;
GET
END_GET
END_PROPERTY

END_INTERFACE

// 40 Visualizations/ABB/580/DIA_ABB580
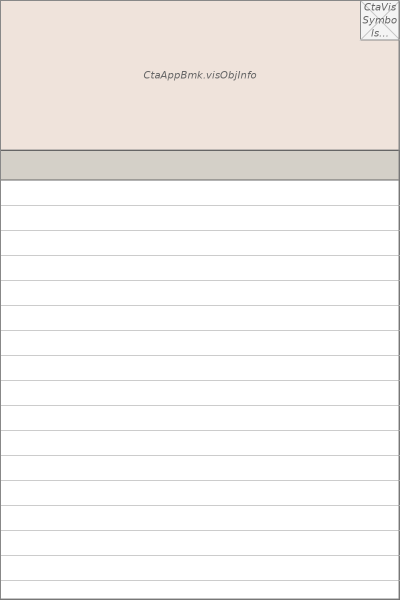
VISUALIZATION DIA_ABB580  // 400x600
VAR_INPUT
	ITF_FU_BASE_IN		: CtaSysFU.ITF_FU_BASE;
END_VAR
VAR
	ITF_FU_ABB_580_QUERRY	:	ITF_FU_ABB_580;
END_VAR
    Rectangle (0,0 400x600)
    Frame (0,0 400x150)
        shows CtaAppBmk.visObjInfo(ITF_BMK_IN := ITF_FU_BASE_IN)
    Frame (0,150 400x450), invisible if: NOT __QUERYINTERFACE(ITF_FU_BASE_IN,ITF_FU_ABB_580_QUERRY)
        shows VIS_ABB580(ITF_FU_ABB_580_IN := ITF_FU_ABB_580_QUERRY)
    Image (360,0 40x40), image: CtaVisSymbols.ImagePool.close_solo_black
        OnMouseClick:  Dialog=Current Dialog, Result=OK, NumpadKeypadSet=True
END_VISUALIZATION

// 40 Visualizations/ABB/580/TABLE/VIS_FU_ABB_TABLE
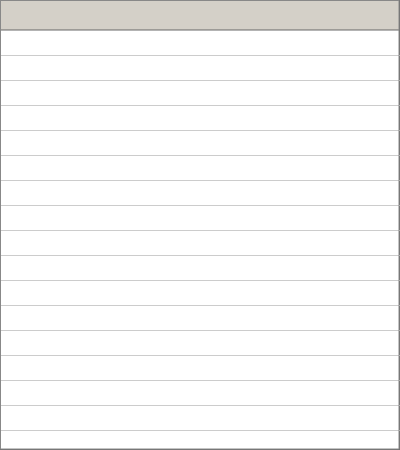
VISUALIZATION VIS_FU_ABB_TABLE  // 400x450
VAR_INPUT	
	ayscTable				:	ARRAY[0..16] OF scFuAbb580Table;
END_VAR
    Table (0,0 400x450), data array: ayscTable
        p1014161805: 16 - 0 + INT#1
        p3854506369: ayscTable[INDEX].stParaNr
        p1892666644: ayscTable[INDEX].stValue
END_VISUALIZATION

// 40 Visualizations/ABB/580/VISU/VIS_ABB580
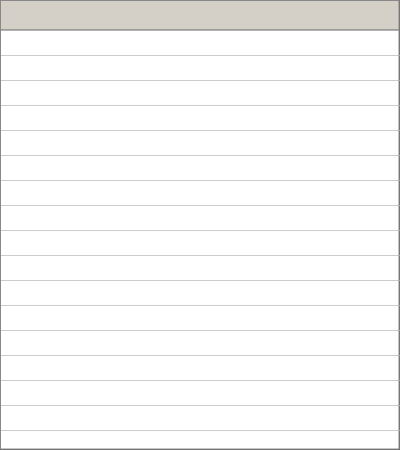
VISUALIZATION VIS_ABB580  // 400x450
VAR_INPUT
	ITF_FU_ABB_580_IN	:	ITF_FU_ABB_580;
END_VAR
    Frame (0,0 400x450), invisible if: NOT __QUERYINTERFACE(ITF_FU_ABB_580_IN,ITF_FU_ABB_580_IN)
        shows VIS_ABB580_QUERY(ITF_FU_ABB_580_IN := ITF_FU_ABB_580_IN)
END_VISUALIZATION

// 40 Visualizations/ABB/580/VISU/VIS_ABB580_QUERY
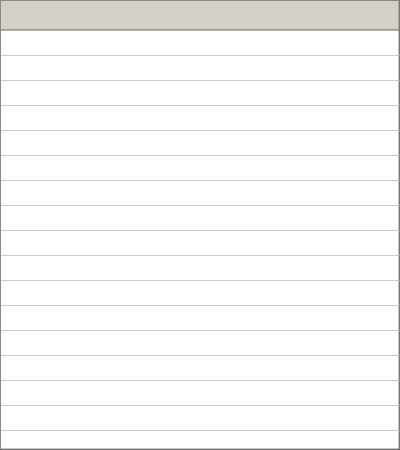
VISUALIZATION VIS_ABB580_QUERY  // 400x450
VAR_INPUT
	ITF_FU_ABB_580_IN	:	ITF_FU_ABB_580;
END_VAR
    Frame (0,0 400x450)
        shows VIS_FU_ABB_TABLE(ayscTable := ITF_FU_ABB_580_IN.proayscTable)
END_VISUALIZATION

// 40 Visualizations/ABB/880/TABLE/VIS_FU_ABB_TABLE_880
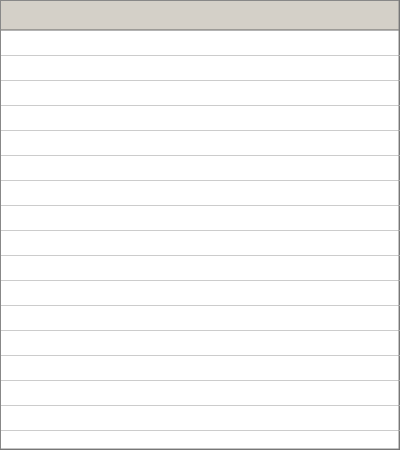
VISUALIZATION VIS_FU_ABB_TABLE_880  // 400x450
VAR_INPUT	
	ayscTable				:	ARRAY[0..16] OF scFuAbb880Table;
END_VAR
    Table (0,0 400x450), data array: ayscTable
        p1014161805: 16 - 0 + INT#1
        p3854506369: ayscTable[INDEX].stParaNr
        p1892666644: ayscTable[INDEX].stValue
END_VISUALIZATION

// 40 Visualizations/ABB/880/VISU/VIS_ABB880
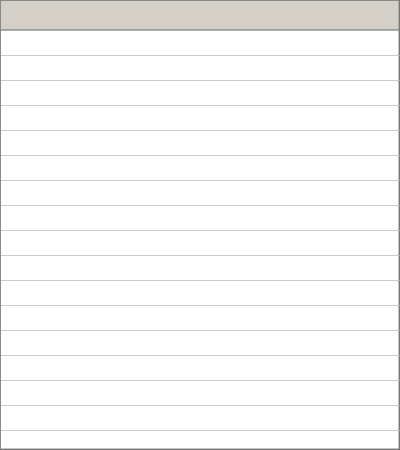
VISUALIZATION VIS_ABB880  // 400x450
VAR_INPUT
	ITF_FU_ABB_880_IN	:	ITF_FU_ABB_880;
END_VAR
    Frame (0,0 400x450), invisible if: NOT __QUERYINTERFACE(ITF_FU_ABB_880_IN,ITF_FU_ABB_880_IN)
        shows VIS_ABB880_QUERY(ITF_FU_ABB_880_IN := ITF_FU_ABB_880_IN)
END_VISUALIZATION

// 40 Visualizations/ABB/880/VISU/VIS_ABB880_QUERY
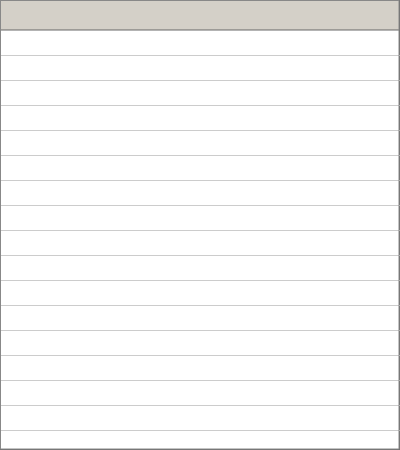
VISUALIZATION VIS_ABB880_QUERY  // 400x450
VAR_INPUT
	ITF_FU_ABB_880_IN	:	ITF_FU_ABB_880;
END_VAR
    Frame (0,0 400x450)
        shows VIS_FU_ABB_TABLE_880(ayscTable := ITF_FU_ABB_880_IN.proayscTable)
END_VISUALIZATION

// 40 Visualizations/ABB/880/DIA_ABB880
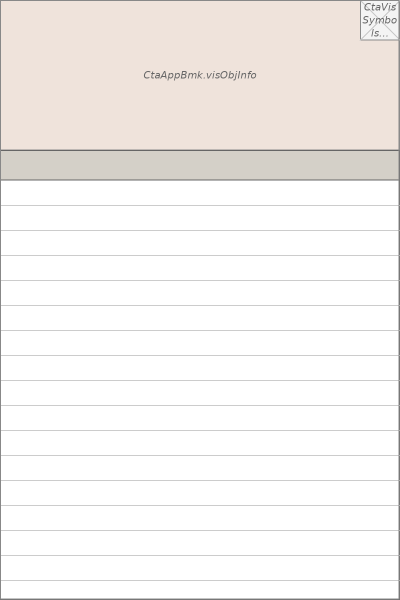
VISUALIZATION DIA_ABB880  // 400x600
VAR_INPUT
	ITF_FU_BASE_IN		: CtaSysFU.ITF_FU_BASE;
END_VAR
VAR
	ITF_FU_ABB_880_QUERRY	:	ITF_FU_ABB_880;
END_VAR
    Rectangle (0,0 400x600)
    Frame (0,0 400x150)
        shows CtaAppBmk.visObjInfo(ITF_BMK_IN := ITF_FU_BASE_IN)
    Frame (0,150 400x450), invisible if: NOT __QUERYINTERFACE(ITF_FU_BASE_IN,ITF_FU_ABB_880_QUERRY)
        shows VIS_ABB880(ITF_FU_ABB_880_IN := ITF_FU_ABB_880_QUERRY)
    Image (360,0 40x40), image: CtaVisSymbols.ImagePool.close_solo_black
        OnMouseClick:  Dialog=Current Dialog, Result=OK, NumpadKeypadSet=True
END_VISUALIZATION

// 40 Visualizations/BITZER/CSV/TABLE/VIS_FU_BITZER_TABLE
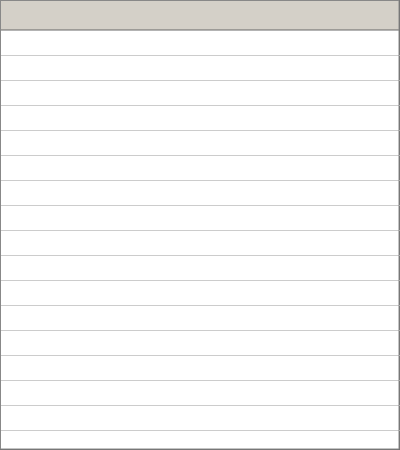
VISUALIZATION VIS_FU_BITZER_TABLE  // 400x450
VAR_INPUT	
	ayscTable				:	ARRAY[0..17] OF scFuBitzerCSVTable;
END_VAR
    Table (0,0 400x450), data array: ayscTable
        p1014161805: 17 - 0 + INT#1
        p3854506369: ayscTable[INDEX].stParaNr
        p1892666644: ayscTable[INDEX].stValue
END_VISUALIZATION

// 40 Visualizations/BITZER/CSV/VISU/VIS_BITZER_CSV
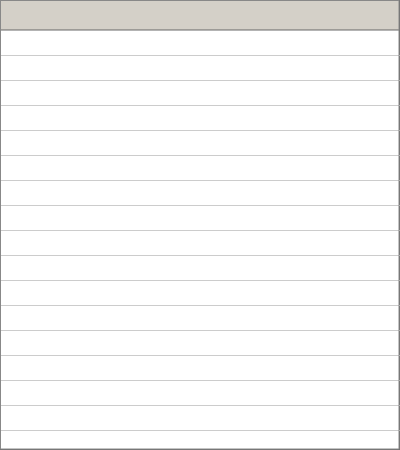
VISUALIZATION VIS_BITZER_CSV  // 400x450
VAR_INPUT
	ITF_FU_BITZER_CSV_IN	:	ITF_FU_BITZER_CSV;
END_VAR
    Frame (0,0 400x450), invisible if: NOT __QUERYINTERFACE(ITF_FU_BITZER_CSV_IN,ITF_FU_BITZER_CSV_IN)
        shows VIS_BITZER_CSV_QUERY(ITF_FU_BITZER_CSV_IN := ITF_FU_BITZER_CSV_IN)
END_VISUALIZATION

// 40 Visualizations/BITZER/CSV/VISU/VIS_BITZER_CSV_QUERY
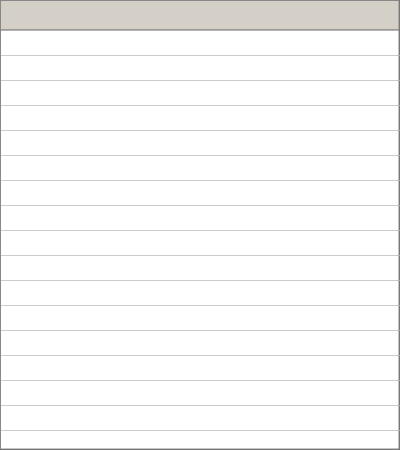
VISUALIZATION VIS_BITZER_CSV_QUERY  // 400x450
VAR_INPUT
	ITF_FU_BITZER_CSV_IN	:	ITF_FU_BITZER_CSV;
END_VAR
    Frame (0,0 400x450)
        shows VIS_FU_BITZER_TABLE(ayscTable := ITF_FU_BITZER_CSV_IN.proayscTable)
END_VISUALIZATION

// 40 Visualizations/BITZER/CSV/DIA_BITZER_CSV
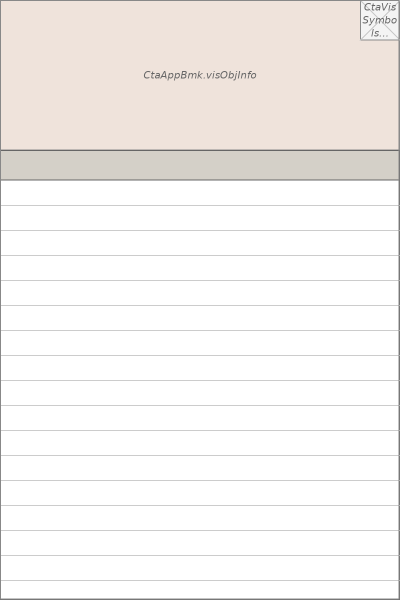
VISUALIZATION DIA_BITZER_CSV  // 400x600
VAR_INPUT
	ITF_FU_BASE_IN		: CtaSysFU.ITF_FU_BASE;
END_VAR
VAR
	ITF_FU_BITZER_CSV_QUERRY	:	ITF_FU_BITZER_CSV;
END_VAR
    Rectangle (0,0 400x600)
    Frame (0,0 400x150)
        shows CtaAppBmk.visObjInfo(ITF_BMK_IN := ITF_FU_BASE_IN)
    Frame (0,150 400x450), invisible if: NOT __QUERYINTERFACE(ITF_FU_BASE_IN,ITF_FU_BITZER_CSV_QUERRY)
        shows VIS_BITZER_CSV(ITF_FU_BITZER_CSV_IN := ITF_FU_BITZER_CSV_QUERRY)
    Image (360,0 40x40), image: CtaVisSymbols.ImagePool.close_solo_black
        OnMouseClick:  Dialog=Current Dialog, Result=OK, NumpadKeypadSet=True
END_VISUALIZATION

(* text list Error_ABB580_880 (id | default | de | en | fr | it)
  20 | Modbus ausfall | Modbus ausfall | Modbus failure | Défaillance Modbus | Errore Modbus
  21 | Modbus Software Time Out | Modbus Software Time Out | Modbus software timeout | Temporisation du logiciel Modbus | Timeout del software Modbus
  22 | FU error:  | FU error:  | FU error:  | FU error:  | FU error: 
   |  |  |  |  |  *)

(* text list Info_ABB580_880 (id | default | de | en | fr | it)
  0 | keine Meldung Anstehend | keine Meldung Anstehend | no message pending | aucun message en attente | nessun messaggio in sospeso
   |  |  |  |  |  *)

(* text list Warnung_ABB580_880 (id | default | de | en | fr | it)
  20 | Firmware Missmatch. Expect:  | Firmware Missmatch. Expect:  | Firmware Missmatch. Expect:  | Firmware Missmatch. Expect:  | 
   |  |  |  |  |  *)

(* text list FU_ABB_580_880_PARA (id | default)
  00.04 | Status Word
  00.05 | Status Wert
  01.06 | Aktuelle Hz
  01.07 | Aktuelle Ampere
  01.13 | Aktuelle Spannung
  01.14 | Aktuelle Leistung 
  01.18 | GWh
  01.19 | MWh
  01.20 | KWh
  04.01 | Fehler Aktuell
  04.02 | Fehler Alt 1
  04.03 | Fehler Alt 2
  05.10 | Temperatur
  05.81 | Frequenz bei Fehler
  05.87 | Temperatur bei Fehler
  30.13 | Min Hz
  46.02 | Max Hz
   |  *)

(* text list Error_BITZER_CSV (id | default | de | en | fr | it)
  20 | Modbus ausfall | Modbus ausfall | Modbus failure | Défaillance Modbus | Errore Modbus
  21 | Modbus Software Time Out | Modbus Software Time Out | Modbus software timeout | Temporisation du logiciel Modbus | Timeout del software Modbus
  22 | FU error:  | FU error:  | FU error:  | FU error:  | FU error: 
   |  |  |  |  |  *)

(* text list Info_BITZER_CSV (id | default | de | en | fr | it)
  0 | keine Meldung Anstehend | keine Meldung Anstehend | no message pending | aucun message en attente | nessun messaggio in sospeso
   |  |  |  |  |  *)

(* text list Warnung_BITZER_CSV (id | default | de | en | fr | it)
  20 | Firmware Missmatch. Expect:  | Firmware Missmatch. Expect:  | Firmware Missmatch. Expect:  | Firmware Missmatch. Expect:  | 
   |  |  |  |  |  *)

(* text list FU_BITZER_CSV_PARA (id | default)
  1 | Aktueller Sollwert
  2 | Aktueller Istwert
  3 | Aktuelle Motordrezahl
  4 | Aktuelles Statusword
  5 | Aktive Störung
  6 | Aktive kritische Meldung
  7 | Aktive Warnung
  8 | Status FU
  9 | Status Antrieb
  10 | Status Einsatzgrenze
  11 | Verdampfungsdruck
  12 | Verdampfungstemperatur
  13 | Verflüssigungsdruck
  14 | Verflüssigungstemperatur
  15 | Öltemperatur
  16 | Motortemperatur
  17 | IGBT- Temperatur
  18 | Kühlplattentemperatur
   |  *)
